// TIA Portal V19 export
DATA_BLOCK "HW_Const_Values"   // DB200
// stored: Access Published, MemoryReserve 100
   VAR
      CU2_PN_IODevice { ExternalAccessible := 'False'; ExternalVisible := 'False'; ExternalWritable := 'False'} : HW_DEVICE := 267;   // "CU2~PN~IODevice"
      CU2_PN { ExternalAccessible := 'False'; ExternalVisible := 'False'; ExternalWritable := 'False'} : HW_INTERFACE := 269;   // "CU2~PN"
      CU2_PN_Port_1 { ExternalAccessible := 'False'; ExternalVisible := 'False'; ExternalWritable := 'False'} : HW_INTERFACE := 270;   // "CU2~PN~Port_1"
      CU2_PN_Port_2 { ExternalAccessible := 'False'; ExternalVisible := 'False'; ExternalWritable := 'False'} : HW_INTERFACE := 271;   // "CU2~PN~Port_2"
      CU2_PN_585A1_ModuleAccessPoint { ExternalAccessible := 'False'; ExternalVisible := 'False'; ExternalWritable := 'False'} : HW_SUBMODULE := 273;   // "CU2~PN~585A1_ModuleAccessPoint"
      CU2_PN_1190A1_ModuleAccessPoint { ExternalAccessible := 'False'; ExternalVisible := 'False'; ExternalWritable := 'False'} : HW_SUBMODULE := 289;   // "CU2~PN~1190A1_ModuleAccessPoint"
      CU2_PN_1300A1_ModuleAccessPoint { ExternalAccessible := 'False'; ExternalVisible := 'False'; ExternalWritable := 'False'} : HW_SUBMODULE := 293;   // "CU2~PN~1300A1_ModuleAccessPoint"
      CU2_PN_830A1_ModuleAccessPoint { ExternalAccessible := 'False'; ExternalVisible := 'False'; ExternalWritable := 'False'} : HW_SUBMODULE := 297;   // "CU2~PN~830A1_ModuleAccessPoint"
      CU2_PN_1 { ExternalAccessible := 'False'; ExternalVisible := 'False'; ExternalWritable := 'False'} : HW_INTERFACE := 269;   // "CU2~PN(1)"
      CU2_PN_Port_1_1 { ExternalAccessible := 'False'; ExternalVisible := 'False'; ExternalWritable := 'False'} : HW_INTERFACE := 270;   // "CU2~PN~Port_1(1)"
      CU2_PN_Port_2_1 { ExternalAccessible := 'False'; ExternalVisible := 'False'; ExternalWritable := 'False'} : HW_INTERFACE := 271;   // "CU2~PN~Port_2(1)"
      CU2_PN_2 { ExternalAccessible := 'False'; ExternalVisible := 'False'; ExternalWritable := 'False'} : HW_INTERFACE := 269;   // "CU2~PN(2)"
      CU2_PN_Port_1_2 { ExternalAccessible := 'False'; ExternalVisible := 'False'; ExternalWritable := 'False'} : HW_INTERFACE := 270;   // "CU2~PN~Port_1(2)"
      CU2_PN_Port_2_2 { ExternalAccessible := 'False'; ExternalVisible := 'False'; ExternalWritable := 'False'} : HW_INTERFACE := 271;   // "CU2~PN~Port_2(2)"
      CU2_PN_3 { ExternalAccessible := 'False'; ExternalVisible := 'False'; ExternalWritable := 'False'} : HW_INTERFACE := 269;   // "CU2~PN(3)"
      CU2_PN_Port_1_3 { ExternalAccessible := 'False'; ExternalVisible := 'False'; ExternalWritable := 'False'} : HW_INTERFACE := 270;   // "CU2~PN~Port_1(3)"
      CU2_PN_Port_2_3 { ExternalAccessible := 'False'; ExternalVisible := 'False'; ExternalWritable := 'False'} : HW_INTERFACE := 271;   // "CU2~PN~Port_2(3)"
      Local_PROFINET_interface_GBIT_3 { ExternalAccessible := 'False'; ExternalVisible := 'False'; ExternalWritable := 'False'} : HW_INTERFACE := 120;   // "Local~PROFINET_interface_GBIT_3"
      Local_PROFINET_interface_GBIT_3_Port_1 { ExternalAccessible := 'False'; ExternalVisible := 'False'; ExternalWritable := 'False'} : HW_INTERFACE := 121;   // "Local~PROFINET_interface_GBIT_3~Port_1"
      Local_412A1 { ExternalAccessible := 'False'; ExternalVisible := 'False'; ExternalWritable := 'False'} : HW_SUBMODULE := 257;   // "Local~412A1"
      Local_413A1 { ExternalAccessible := 'False'; ExternalVisible := 'False'; ExternalWritable := 'False'} : HW_SUBMODULE := 258;   // "Local~413A1"
      Local_413A2 { ExternalAccessible := 'False'; ExternalVisible := 'False'; ExternalWritable := 'False'} : HW_SUBMODULE := 259;   // "Local~413A2"
      Local_414A1 { ExternalAccessible := 'False'; ExternalVisible := 'False'; ExternalWritable := 'False'} : HW_SUBMODULE := 260;   // "Local~414A1"
      Local_415A1 { ExternalAccessible := 'False'; ExternalVisible := 'False'; ExternalWritable := 'False'} : HW_SUBMODULE := 261;   // "Local~415A1"
      Local_415A2 { ExternalAccessible := 'False'; ExternalVisible := 'False'; ExternalWritable := 'False'} : HW_SUBMODULE := 263;   // "Local~415A2"
      HW_460A1_JB001_Proxy { ExternalAccessible := 'False'; ExternalVisible := 'False'; ExternalWritable := 'False'} : HW_SUBMODULE := 302;   // "460A1_JB001~Proxy"
      HW_460A1_JB001_IODevice { ExternalAccessible := 'False'; ExternalVisible := 'False'; ExternalWritable := 'False'} : HW_DEVICE := 300;   // "460A1_JB001~IODevice"
      HW_460A1_JB001_Head { ExternalAccessible := 'False'; ExternalVisible := 'False'; ExternalWritable := 'False'} : HW_SUBMODULE := 303;   // "460A1_JB001~Head"
      HW_460A1_JB001_460A1_X1 { ExternalAccessible := 'False'; ExternalVisible := 'False'; ExternalWritable := 'False'} : HW_INTERFACE := 304;   // "460A1_JB001~460A1_X1"
      HW_460A1_JB001_479A3 { ExternalAccessible := 'False'; ExternalVisible := 'False'; ExternalWritable := 'False'} : HW_SUBMODULE := 355;   // "460A1_JB001~479A3"
      HW_460A1_JB001_479A4 { ExternalAccessible := 'False'; ExternalVisible := 'False'; ExternalWritable := 'False'} : HW_SUBMODULE := 356;   // "460A1_JB001~479A4"
      HW_460A1_JB001_480A1 { ExternalAccessible := 'False'; ExternalVisible := 'False'; ExternalWritable := 'False'} : HW_SUBMODULE := 357;   // "460A1_JB001~480A1"
      HW_460A1_JB001_480A2 { ExternalAccessible := 'False'; ExternalVisible := 'False'; ExternalWritable := 'False'} : HW_SUBMODULE := 358;   // "460A1_JB001~480A2"
      HW_460A1_JB001_482A1 { ExternalAccessible := 'False'; ExternalVisible := 'False'; ExternalWritable := 'False'} : HW_SUBMODULE := 359;   // "460A1_JB001~482A1"
      HW_460A1_JB001_482A2 { ExternalAccessible := 'False'; ExternalVisible := 'False'; ExternalWritable := 'False'} : HW_SUBMODULE := 360;   // "460A1_JB001~482A2"
      HW_460A1_JB001_Server_module_1 { ExternalAccessible := 'False'; ExternalVisible := 'False'; ExternalWritable := 'False'} : HW_SUBMODULE := 456;   // "460A1_JB001~Server_module_1"
      HW_460A1_JB001_464A1 { ExternalAccessible := 'False'; ExternalVisible := 'False'; ExternalWritable := 'False'} : HW_SUBMODULE := 308;   // "460A1_JB001~464A1"
      HW_460A1_JB001_470A2 { ExternalAccessible := 'False'; ExternalVisible := 'False'; ExternalWritable := 'False'} : HW_SUBMODULE := 704;   // "460A1_JB001~470A2"
      HW_460A1_JB001_470A1 { ExternalAccessible := 'False'; ExternalVisible := 'False'; ExternalWritable := 'False'} : HW_SUBMODULE := 703;   // "460A1_JB001~470A1"
      HW_460A1_JB001_463A1 { ExternalAccessible := 'False'; ExternalVisible := 'False'; ExternalWritable := 'False'} : HW_SUBMODULE := 307;   // "460A1_JB001~463A1"
      HW_460A1_JB001_460A1_X1_Port_2 { ExternalAccessible := 'False'; ExternalVisible := 'False'; ExternalWritable := 'False'} : HW_INTERFACE := 306;   // "460A1_JB001~460A1_X1~Port_2"
      HW_460A1_JB001_460A1_X1_Port_1 { ExternalAccessible := 'False'; ExternalVisible := 'False'; ExternalWritable := 'False'} : HW_INTERFACE := 305;   // "460A1_JB001~460A1_X1~Port_1"
      HW_460A1_JB001_465A1 { ExternalAccessible := 'False'; ExternalVisible := 'False'; ExternalWritable := 'False'} : HW_SUBMODULE := 309;   // "460A1_JB001~465A1"
      HW_460A1_JB001_468A1 { ExternalAccessible := 'False'; ExternalVisible := 'False'; ExternalWritable := 'False'} : HW_SUBMODULE := 310;   // "460A1_JB001~468A1"
      HW_460A1_JB001_468A2 { ExternalAccessible := 'False'; ExternalVisible := 'False'; ExternalWritable := 'False'} : HW_SUBMODULE := 311;   // "460A1_JB001~468A2"
      HW_460A1_JB001_468A3 { ExternalAccessible := 'False'; ExternalVisible := 'False'; ExternalWritable := 'False'} : HW_SUBMODULE := 312;   // "460A1_JB001~468A3"
      HW_460A1_JB001_468A4 { ExternalAccessible := 'False'; ExternalVisible := 'False'; ExternalWritable := 'False'} : HW_SUBMODULE := 313;   // "460A1_JB001~468A4"
      HW_460A1_JB001_468A5 { ExternalAccessible := 'False'; ExternalVisible := 'False'; ExternalWritable := 'False'} : HW_SUBMODULE := 314;   // "460A1_JB001~468A5"
      HW_460A1_JB001_468A6 { ExternalAccessible := 'False'; ExternalVisible := 'False'; ExternalWritable := 'False'} : HW_SUBMODULE := 315;   // "460A1_JB001~468A6"
      HW_460A1_JB001_468A7 { ExternalAccessible := 'False'; ExternalVisible := 'False'; ExternalWritable := 'False'} : HW_SUBMODULE := 316;   // "460A1_JB001~468A7"
      HW_460A1_JB001_468A8 { ExternalAccessible := 'False'; ExternalVisible := 'False'; ExternalWritable := 'False'} : HW_SUBMODULE := 317;   // "460A1_JB001~468A8"
      HW_460A1_JB001_471A1 { ExternalAccessible := 'False'; ExternalVisible := 'False'; ExternalWritable := 'False'} : HW_SUBMODULE := 320;   // "460A1_JB001~471A1"
      HW_460A1_JB001_471A2 { ExternalAccessible := 'False'; ExternalVisible := 'False'; ExternalWritable := 'False'} : HW_SUBMODULE := 321;   // "460A1_JB001~471A2"
      HW_460A1_JB001_472A1 { ExternalAccessible := 'False'; ExternalVisible := 'False'; ExternalWritable := 'False'} : HW_SUBMODULE := 322;   // "460A1_JB001~472A1"
      HW_460A1_JB001_474A1 { ExternalAccessible := 'False'; ExternalVisible := 'False'; ExternalWritable := 'False'} : HW_SUBMODULE := 323;   // "460A1_JB001~474A1"
      HW_460A1_JB001_474A2 { ExternalAccessible := 'False'; ExternalVisible := 'False'; ExternalWritable := 'False'} : HW_SUBMODULE := 324;   // "460A1_JB001~474A2"
      HW_460A1_JB001_474A3 { ExternalAccessible := 'False'; ExternalVisible := 'False'; ExternalWritable := 'False'} : HW_SUBMODULE := 325;   // "460A1_JB001~474A3"
      HW_460A1_JB001_474A4 { ExternalAccessible := 'False'; ExternalVisible := 'False'; ExternalWritable := 'False'} : HW_SUBMODULE := 326;   // "460A1_JB001~474A4"
      HW_460A1_JB001_474A5 { ExternalAccessible := 'False'; ExternalVisible := 'False'; ExternalWritable := 'False'} : HW_SUBMODULE := 327;   // "460A1_JB001~474A5"
      HW_460A1_JB001_474A6 { ExternalAccessible := 'False'; ExternalVisible := 'False'; ExternalWritable := 'False'} : HW_SUBMODULE := 328;   // "460A1_JB001~474A6"
      HW_460A1_JB001_474A7 { ExternalAccessible := 'False'; ExternalVisible := 'False'; ExternalWritable := 'False'} : HW_SUBMODULE := 329;   // "460A1_JB001~474A7"
      HW_460A1_JB001_474A8 { ExternalAccessible := 'False'; ExternalVisible := 'False'; ExternalWritable := 'False'} : HW_SUBMODULE := 330;   // "460A1_JB001~474A8"
      HW_460A1_JB001_475A1 { ExternalAccessible := 'False'; ExternalVisible := 'False'; ExternalWritable := 'False'} : HW_SUBMODULE := 331;   // "460A1_JB001~475A1"
      HW_460A1_JB001_475A2 { ExternalAccessible := 'False'; ExternalVisible := 'False'; ExternalWritable := 'False'} : HW_SUBMODULE := 332;   // "460A1_JB001~475A2"
      HW_460A1_JB001_475A3 { ExternalAccessible := 'False'; ExternalVisible := 'False'; ExternalWritable := 'False'} : HW_SUBMODULE := 333;   // "460A1_JB001~475A3"
      HW_460A1_JB001_475A4 { ExternalAccessible := 'False'; ExternalVisible := 'False'; ExternalWritable := 'False'} : HW_SUBMODULE := 334;   // "460A1_JB001~475A4"
      HW_460A1_JB001_475A5 { ExternalAccessible := 'False'; ExternalVisible := 'False'; ExternalWritable := 'False'} : HW_SUBMODULE := 335;   // "460A1_JB001~475A5"
      HW_460A1_JB001_475A6 { ExternalAccessible := 'False'; ExternalVisible := 'False'; ExternalWritable := 'False'} : HW_SUBMODULE := 336;   // "460A1_JB001~475A6"
      HW_460A1_JB001_475A7 { ExternalAccessible := 'False'; ExternalVisible := 'False'; ExternalWritable := 'False'} : HW_SUBMODULE := 337;   // "460A1_JB001~475A7"
      HW_460A1_JB001_475A8 { ExternalAccessible := 'False'; ExternalVisible := 'False'; ExternalWritable := 'False'} : HW_SUBMODULE := 338;   // "460A1_JB001~475A8"
      HW_460A1_JB001_476A1 { ExternalAccessible := 'False'; ExternalVisible := 'False'; ExternalWritable := 'False'} : HW_SUBMODULE := 339;   // "460A1_JB001~476A1"
      HW_460A1_JB001_476A2 { ExternalAccessible := 'False'; ExternalVisible := 'False'; ExternalWritable := 'False'} : HW_SUBMODULE := 340;   // "460A1_JB001~476A2"
      HW_460A1_JB001_476A3 { ExternalAccessible := 'False'; ExternalVisible := 'False'; ExternalWritable := 'False'} : HW_SUBMODULE := 341;   // "460A1_JB001~476A3"
      HW_460A1_JB001_476A4 { ExternalAccessible := 'False'; ExternalVisible := 'False'; ExternalWritable := 'False'} : HW_SUBMODULE := 342;   // "460A1_JB001~476A4"
      HW_460A1_JB001_476A5 { ExternalAccessible := 'False'; ExternalVisible := 'False'; ExternalWritable := 'False'} : HW_SUBMODULE := 343;   // "460A1_JB001~476A5"
      HW_460A1_JB001_476A6 { ExternalAccessible := 'False'; ExternalVisible := 'False'; ExternalWritable := 'False'} : HW_SUBMODULE := 344;   // "460A1_JB001~476A6"
      HW_460A1_JB001_478A1 { ExternalAccessible := 'False'; ExternalVisible := 'False'; ExternalWritable := 'False'} : HW_SUBMODULE := 345;   // "460A1_JB001~478A1"
      HW_460A1_JB001_478A2 { ExternalAccessible := 'False'; ExternalVisible := 'False'; ExternalWritable := 'False'} : HW_SUBMODULE := 346;   // "460A1_JB001~478A2"
      HW_460A1_JB001_478A3 { ExternalAccessible := 'False'; ExternalVisible := 'False'; ExternalWritable := 'False'} : HW_SUBMODULE := 347;   // "460A1_JB001~478A3"
      HW_460A1_JB001_478A4 { ExternalAccessible := 'False'; ExternalVisible := 'False'; ExternalWritable := 'False'} : HW_SUBMODULE := 348;   // "460A1_JB001~478A4"
      HW_460A1_JB001_478A5 { ExternalAccessible := 'False'; ExternalVisible := 'False'; ExternalWritable := 'False'} : HW_SUBMODULE := 349;   // "460A1_JB001~478A5"
      HW_460A1_JB001_478A6 { ExternalAccessible := 'False'; ExternalVisible := 'False'; ExternalWritable := 'False'} : HW_SUBMODULE := 350;   // "460A1_JB001~478A6"
      HW_460A1_JB001_478A7 { ExternalAccessible := 'False'; ExternalVisible := 'False'; ExternalWritable := 'False'} : HW_SUBMODULE := 351;   // "460A1_JB001~478A7"
      HW_460A1_JB001_478A8 { ExternalAccessible := 'False'; ExternalVisible := 'False'; ExternalWritable := 'False'} : HW_SUBMODULE := 352;   // "460A1_JB001~478A8"
      HW_460A1_JB001_479A1 { ExternalAccessible := 'False'; ExternalVisible := 'False'; ExternalWritable := 'False'} : HW_SUBMODULE := 353;   // "460A1_JB001~479A1"
      HW_460A1_JB001_479A2 { ExternalAccessible := 'False'; ExternalVisible := 'False'; ExternalWritable := 'False'} : HW_SUBMODULE := 354;   // "460A1_JB001~479A2"
      HW_490A1_JB301_Proxy { ExternalAccessible := 'False'; ExternalVisible := 'False'; ExternalWritable := 'False'} : HW_SUBMODULE := 363;   // "490A1_JB301~Proxy"
      HW_490A1_JB301_IODevice { ExternalAccessible := 'False'; ExternalVisible := 'False'; ExternalWritable := 'False'} : HW_DEVICE := 361;   // "490A1_JB301~IODevice"
      HW_490A1_JB301_Head { ExternalAccessible := 'False'; ExternalVisible := 'False'; ExternalWritable := 'False'} : HW_SUBMODULE := 364;   // "490A1_JB301~Head"
      HW_490A1_JB301_PROFINET_interface { ExternalAccessible := 'False'; ExternalVisible := 'False'; ExternalWritable := 'False'} : HW_INTERFACE := 365;   // "490A1_JB301~PROFINET_interface"
      HW_490A1_JB301_495A2 { ExternalAccessible := 'False'; ExternalVisible := 'False'; ExternalWritable := 'False'} : HW_SUBMODULE := 369;   // "490A1_JB301~495A2"
      HW_490A1_JB301_495A1 { ExternalAccessible := 'False'; ExternalVisible := 'False'; ExternalWritable := 'False'} : HW_SUBMODULE := 368;   // "490A1_JB301~495A1"
      HW_490A1_JB301_PROFINET_interface_Port_2 { ExternalAccessible := 'False'; ExternalVisible := 'False'; ExternalWritable := 'False'} : HW_INTERFACE := 367;   // "490A1_JB301~PROFINET_interface~Port_2"
      HW_490A1_JB301_PROFINET_interface_Port_1 { ExternalAccessible := 'False'; ExternalVisible := 'False'; ExternalWritable := 'False'} : HW_INTERFACE := 366;   // "490A1_JB301~PROFINET_interface~Port_1"
      HW_510A1_JB302_Proxy { ExternalAccessible := 'False'; ExternalVisible := 'False'; ExternalWritable := 'False'} : HW_SUBMODULE := 378;   // "510A1_JB302~Proxy"
      HW_510A1_JB302_IODevice { ExternalAccessible := 'False'; ExternalVisible := 'False'; ExternalWritable := 'False'} : HW_DEVICE := 376;   // "510A1_JB302~IODevice"
      HW_510A1_JB302_Head { ExternalAccessible := 'False'; ExternalVisible := 'False'; ExternalWritable := 'False'} : HW_SUBMODULE := 379;   // "510A1_JB302~Head"
      HW_510A1_JB302_PROFINET_interface { ExternalAccessible := 'False'; ExternalVisible := 'False'; ExternalWritable := 'False'} : HW_INTERFACE := 380;   // "510A1_JB302~PROFINET_interface"
      HW_510A1_JB302_515A2 { ExternalAccessible := 'False'; ExternalVisible := 'False'; ExternalWritable := 'False'} : HW_SUBMODULE := 386;   // "510A1_JB302~515A2"
      HW_510A1_JB302_515A1 { ExternalAccessible := 'False'; ExternalVisible := 'False'; ExternalWritable := 'False'} : HW_SUBMODULE := 385;   // "510A1_JB302~515A1"
      HW_510A1_JB302_513A1 { ExternalAccessible := 'False'; ExternalVisible := 'False'; ExternalWritable := 'False'} : HW_SUBMODULE := 384;   // "510A1_JB302~513A1"
      HW_510A1_JB302_512A1 { ExternalAccessible := 'False'; ExternalVisible := 'False'; ExternalWritable := 'False'} : HW_SUBMODULE := 383;   // "510A1_JB302~512A1"
      HW_510A1_JB302_PROFINET_interface_Port_2 { ExternalAccessible := 'False'; ExternalVisible := 'False'; ExternalWritable := 'False'} : HW_INTERFACE := 382;   // "510A1_JB302~PROFINET_interface~Port_2"
      HW_510A1_JB302_PROFINET_interface_Port_1 { ExternalAccessible := 'False'; ExternalVisible := 'False'; ExternalWritable := 'False'} : HW_INTERFACE := 381;   // "510A1_JB302~PROFINET_interface~Port_1"
      HW_530A1_JB305_Proxy { ExternalAccessible := 'False'; ExternalVisible := 'False'; ExternalWritable := 'False'} : HW_SUBMODULE := 413;   // "530A1_JB305~Proxy"
      HW_530A1_JB305_IODevice { ExternalAccessible := 'False'; ExternalVisible := 'False'; ExternalWritable := 'False'} : HW_DEVICE := 411;   // "530A1_JB305~IODevice"
      HW_530A1_JB305_Head { ExternalAccessible := 'False'; ExternalVisible := 'False'; ExternalWritable := 'False'} : HW_SUBMODULE := 414;   // "530A1_JB305~Head"
      HW_530A1_JB305_PROFINET_interface { ExternalAccessible := 'False'; ExternalVisible := 'False'; ExternalWritable := 'False'} : HW_INTERFACE := 415;   // "530A1_JB305~PROFINET_interface"
      HW_530A1_JB305_542A3 { ExternalAccessible := 'False'; ExternalVisible := 'False'; ExternalWritable := 'False'} : HW_SUBMODULE := 434;   // "530A1_JB305~542A3"
      HW_530A1_JB305_542A2 { ExternalAccessible := 'False'; ExternalVisible := 'False'; ExternalWritable := 'False'} : HW_SUBMODULE := 433;   // "530A1_JB305~542A2"
      HW_530A1_JB305_542A1 { ExternalAccessible := 'False'; ExternalVisible := 'False'; ExternalWritable := 'False'} : HW_SUBMODULE := 432;   // "530A1_JB305~542A1"
      HW_530A1_JB305_540A2 { ExternalAccessible := 'False'; ExternalVisible := 'False'; ExternalWritable := 'False'} : HW_SUBMODULE := 431;   // "530A1_JB305~540A2"
      HW_530A1_JB305_540A1 { ExternalAccessible := 'False'; ExternalVisible := 'False'; ExternalWritable := 'False'} : HW_SUBMODULE := 430;   // "530A1_JB305~540A1"
      HW_530A1_JB305_538A6 { ExternalAccessible := 'False'; ExternalVisible := 'False'; ExternalWritable := 'False'} : HW_SUBMODULE := 429;   // "530A1_JB305~538A6"
      HW_530A1_JB305_538A5 { ExternalAccessible := 'False'; ExternalVisible := 'False'; ExternalWritable := 'False'} : HW_SUBMODULE := 428;   // "530A1_JB305~538A5"
      HW_530A1_JB305_538A4 { ExternalAccessible := 'False'; ExternalVisible := 'False'; ExternalWritable := 'False'} : HW_SUBMODULE := 427;   // "530A1_JB305~538A4"
      HW_530A1_JB305_538A3 { ExternalAccessible := 'False'; ExternalVisible := 'False'; ExternalWritable := 'False'} : HW_SUBMODULE := 426;   // "530A1_JB305~538A3"
      HW_530A1_JB305_538A2 { ExternalAccessible := 'False'; ExternalVisible := 'False'; ExternalWritable := 'False'} : HW_SUBMODULE := 425;   // "530A1_JB305~538A2"
      HW_530A1_JB305_538A1 { ExternalAccessible := 'False'; ExternalVisible := 'False'; ExternalWritable := 'False'} : HW_SUBMODULE := 424;   // "530A1_JB305~538A1"
      HW_530A1_JB305_537A1 { ExternalAccessible := 'False'; ExternalVisible := 'False'; ExternalWritable := 'False'} : HW_SUBMODULE := 423;   // "530A1_JB305~537A1"
      HW_530A1_JB305_536A1 { ExternalAccessible := 'False'; ExternalVisible := 'False'; ExternalWritable := 'False'} : HW_SUBMODULE := 422;   // "530A1_JB305~536A1"
      HW_530A1_JB305_535A2 { ExternalAccessible := 'False'; ExternalVisible := 'False'; ExternalWritable := 'False'} : HW_SUBMODULE := 421;   // "530A1_JB305~535A2"
      HW_530A1_JB305_535A1 { ExternalAccessible := 'False'; ExternalVisible := 'False'; ExternalWritable := 'False'} : HW_SUBMODULE := 420;   // "530A1_JB305~535A1"
      HW_530A1_JB305_533A1 { ExternalAccessible := 'False'; ExternalVisible := 'False'; ExternalWritable := 'False'} : HW_SUBMODULE := 419;   // "530A1_JB305~533A1"
      HW_530A1_JB305_PROFINET_interface_Port_2 { ExternalAccessible := 'False'; ExternalVisible := 'False'; ExternalWritable := 'False'} : HW_INTERFACE := 417;   // "530A1_JB305~PROFINET_interface~Port_2"
      HW_530A1_JB305_PROFINET_interface_Port_1 { ExternalAccessible := 'False'; ExternalVisible := 'False'; ExternalWritable := 'False'} : HW_INTERFACE := 416;   // "530A1_JB305~PROFINET_interface~Port_1"
      HW_550A1_JB306_Proxy { ExternalAccessible := 'False'; ExternalVisible := 'False'; ExternalWritable := 'False'} : HW_SUBMODULE := 437;   // "550A1_JB306~Proxy"
      HW_550A1_JB306_IODevice { ExternalAccessible := 'False'; ExternalVisible := 'False'; ExternalWritable := 'False'} : HW_DEVICE := 435;   // "550A1_JB306~IODevice"
      HW_550A1_JB306_Head { ExternalAccessible := 'False'; ExternalVisible := 'False'; ExternalWritable := 'False'} : HW_SUBMODULE := 438;   // "550A1_JB306~Head"
      HW_550A1_JB306_PROFINET_interface { ExternalAccessible := 'False'; ExternalVisible := 'False'; ExternalWritable := 'False'} : HW_INTERFACE := 439;   // "550A1_JB306~PROFINET_interface"
      HW_550A1_JB306_562A3 { ExternalAccessible := 'False'; ExternalVisible := 'False'; ExternalWritable := 'False'} : HW_SUBMODULE := 455;   // "550A1_JB306~562A3"
      HW_550A1_JB306_562A2 { ExternalAccessible := 'False'; ExternalVisible := 'False'; ExternalWritable := 'False'} : HW_SUBMODULE := 454;   // "550A1_JB306~562A2"
      HW_550A1_JB306_562A1 { ExternalAccessible := 'False'; ExternalVisible := 'False'; ExternalWritable := 'False'} : HW_SUBMODULE := 453;   // "550A1_JB306~562A1"
      HW_550A1_JB306_560A2 { ExternalAccessible := 'False'; ExternalVisible := 'False'; ExternalWritable := 'False'} : HW_SUBMODULE := 452;   // "550A1_JB306~560A2"
      HW_550A1_JB306_560A1 { ExternalAccessible := 'False'; ExternalVisible := 'False'; ExternalWritable := 'False'} : HW_SUBMODULE := 451;   // "550A1_JB306~560A1"
      HW_550A1_JB306_558A6 { ExternalAccessible := 'False'; ExternalVisible := 'False'; ExternalWritable := 'False'} : HW_SUBMODULE := 450;   // "550A1_JB306~558A6"
      HW_550A1_JB306_558A5 { ExternalAccessible := 'False'; ExternalVisible := 'False'; ExternalWritable := 'False'} : HW_SUBMODULE := 449;   // "550A1_JB306~558A5"
      HW_550A1_JB306_558A4 { ExternalAccessible := 'False'; ExternalVisible := 'False'; ExternalWritable := 'False'} : HW_SUBMODULE := 448;   // "550A1_JB306~558A4"
      HW_550A1_JB306_558A3 { ExternalAccessible := 'False'; ExternalVisible := 'False'; ExternalWritable := 'False'} : HW_SUBMODULE := 447;   // "550A1_JB306~558A3"
      HW_550A1_JB306_558A2 { ExternalAccessible := 'False'; ExternalVisible := 'False'; ExternalWritable := 'False'} : HW_SUBMODULE := 446;   // "550A1_JB306~558A2"
      HW_550A1_JB306_558A1 { ExternalAccessible := 'False'; ExternalVisible := 'False'; ExternalWritable := 'False'} : HW_SUBMODULE := 445;   // "550A1_JB306~558A1"
      HW_550A1_JB306_556A1 { ExternalAccessible := 'False'; ExternalVisible := 'False'; ExternalWritable := 'False'} : HW_SUBMODULE := 444;   // "550A1_JB306~556A1"
      HW_550A1_JB306_555A1 { ExternalAccessible := 'False'; ExternalVisible := 'False'; ExternalWritable := 'False'} : HW_SUBMODULE := 443;   // "550A1_JB306~555A1"
      HW_550A1_JB306_552A1 { ExternalAccessible := 'False'; ExternalVisible := 'False'; ExternalWritable := 'False'} : HW_SUBMODULE := 442;   // "550A1_JB306~552A1"
      HW_550A1_JB306_PROFINET_interface_Port_2 { ExternalAccessible := 'False'; ExternalVisible := 'False'; ExternalWritable := 'False'} : HW_INTERFACE := 441;   // "550A1_JB306~PROFINET_interface~Port_2"
      HW_550A1_JB306_PROFINET_interface_Port_1 { ExternalAccessible := 'False'; ExternalVisible := 'False'; ExternalWritable := 'False'} : HW_INTERFACE := 440;   // "550A1_JB306~PROFINET_interface~Port_1"
      CU1_PN_IODevice { ExternalAccessible := 'False'; ExternalVisible := 'False'; ExternalWritable := 'False'} : HW_DEVICE := 275;   // "CU1~PN~IODevice"
      CU1_PN { ExternalAccessible := 'False'; ExternalVisible := 'False'; ExternalWritable := 'False'} : HW_INTERFACE := 277;   // "CU1~PN"
      CU1_PN_Port_1 { ExternalAccessible := 'False'; ExternalVisible := 'False'; ExternalWritable := 'False'} : HW_INTERFACE := 278;   // "CU1~PN~Port_1"
      CU1_PN_Port_2 { ExternalAccessible := 'False'; ExternalVisible := 'False'; ExternalWritable := 'False'} : HW_INTERFACE := 279;   // "CU1~PN~Port_2"
      CU1_PN_580A1_ModuleAccessPoint { ExternalAccessible := 'False'; ExternalVisible := 'False'; ExternalWritable := 'False'} : HW_SUBMODULE := 281;   // "CU1~PN~580A1_ModuleAccessPoint"
      CU1_PN_740A1_1_ModuleAccessPoint { ExternalAccessible := 'False'; ExternalVisible := 'False'; ExternalWritable := 'False'} : HW_SUBMODULE := 284;   // "CU1~PN~740A1_1_ModuleAccessPoint"
      CU1_PN_740A1_2_ModuleAccessPoint { ExternalAccessible := 'False'; ExternalVisible := 'False'; ExternalWritable := 'False'} : HW_SUBMODULE := 318;   // "CU1~PN~740A1_2_ModuleAccessPoint"
      CU1_PN_690A1_1_ModuleAccessPoint { ExternalAccessible := 'False'; ExternalVisible := 'False'; ExternalWritable := 'False'} : HW_SUBMODULE := 459;   // "CU1~PN~690A1_1_ModuleAccessPoint"
      CU1_PN_690A1_2_ModuleAccessPoint { ExternalAccessible := 'False'; ExternalVisible := 'False'; ExternalWritable := 'False'} : HW_SUBMODULE := 463;   // "CU1~PN~690A1_2_ModuleAccessPoint"
      CU1_PN_890A1_1_ModuleAccessPoint { ExternalAccessible := 'False'; ExternalVisible := 'False'; ExternalWritable := 'False'} : HW_SUBMODULE := 467;   // "CU1~PN~890A1_1_ModuleAccessPoint"
      CU1_PN_890A1_2_ModuleAccessPoint { ExternalAccessible := 'False'; ExternalVisible := 'False'; ExternalWritable := 'False'} : HW_SUBMODULE := 471;   // "CU1~PN~890A1_2_ModuleAccessPoint"
      CU1_PN_1 { ExternalAccessible := 'False'; ExternalVisible := 'False'; ExternalWritable := 'False'} : HW_INTERFACE := 277;   // "CU1~PN(1)"
      CU1_PN_Port_1_1 { ExternalAccessible := 'False'; ExternalVisible := 'False'; ExternalWritable := 'False'} : HW_INTERFACE := 278;   // "CU1~PN~Port_1(1)"
      CU1_PN_Port_2_1 { ExternalAccessible := 'False'; ExternalVisible := 'False'; ExternalWritable := 'False'} : HW_INTERFACE := 279;   // "CU1~PN~Port_2(1)"
      CU1_PN_2 { ExternalAccessible := 'False'; ExternalVisible := 'False'; ExternalWritable := 'False'} : HW_INTERFACE := 277;   // "CU1~PN(2)"
      CU1_PN_Port_1_2 { ExternalAccessible := 'False'; ExternalVisible := 'False'; ExternalWritable := 'False'} : HW_INTERFACE := 278;   // "CU1~PN~Port_1(2)"
      CU1_PN_Port_2_2 { ExternalAccessible := 'False'; ExternalVisible := 'False'; ExternalWritable := 'False'} : HW_INTERFACE := 279;   // "CU1~PN~Port_2(2)"
      CU1_PN_3 { ExternalAccessible := 'False'; ExternalVisible := 'False'; ExternalWritable := 'False'} : HW_INTERFACE := 277;   // "CU1~PN(3)"
      CU1_PN_Port_1_3 { ExternalAccessible := 'False'; ExternalVisible := 'False'; ExternalWritable := 'False'} : HW_INTERFACE := 278;   // "CU1~PN~Port_1(3)"
      CU1_PN_Port_2_3 { ExternalAccessible := 'False'; ExternalVisible := 'False'; ExternalWritable := 'False'} : HW_INTERFACE := 279;   // "CU1~PN~Port_2(3)"
      CU3_PROFINET_interface_IODevice { ExternalAccessible := 'False'; ExternalVisible := 'False'; ExternalWritable := 'False'} : HW_DEVICE := 475;   // "CU3~PROFINET_interface~IODevice"
      CU3_PROFINET_interface { ExternalAccessible := 'False'; ExternalVisible := 'False'; ExternalWritable := 'False'} : HW_INTERFACE := 477;   // "CU3~PROFINET_interface"
      CU3_PROFINET_interface_Port_1 { ExternalAccessible := 'False'; ExternalVisible := 'False'; ExternalWritable := 'False'} : HW_INTERFACE := 478;   // "CU3~PROFINET_interface~Port_1"
      CU3_PROFINET_interface_Port_2 { ExternalAccessible := 'False'; ExternalVisible := 'False'; ExternalWritable := 'False'} : HW_INTERFACE := 479;   // "CU3~PROFINET_interface~Port_2"
      CU3_PROFINET_interface_590A1_ModuleAccessPoint { ExternalAccessible := 'False'; ExternalVisible := 'False'; ExternalWritable := 'False'} : HW_SUBMODULE := 481;   // "CU3~PROFINET_interface~590A1_ModuleAccessPoint"
      CU3_PROFINET_interface_590A1_SIEMENS_telegram_393 { ExternalAccessible := 'False'; ExternalVisible := 'False'; ExternalWritable := 'False'} : HW_SUBMODULE := 482;   // "CU3~PROFINET_interface~590A1_SIEMENS_telegram_393"
      CU3_PROFINET_interface_1410A1_1_ModuleAccessPoint { ExternalAccessible := 'False'; ExternalVisible := 'False'; ExternalWritable := 'False'} : HW_SUBMODULE := 484;   // "CU3~PROFINET_interface~1410A1_1_ModuleAccessPoint"
      CU3_PROFINET_interface_1410A1_1_PROFIsafe_telegram_30 { ExternalAccessible := 'False'; ExternalVisible := 'False'; ExternalWritable := 'False'} : HW_SUBMODULE := 486;   // "CU3~PROFINET_interface~1410A1_1_PROFIsafe_telegram_30"
      CU3_PROFINET_interface_1410A1_2_ModuleAccessPoint { ExternalAccessible := 'False'; ExternalVisible := 'False'; ExternalWritable := 'False'} : HW_SUBMODULE := 488;   // "CU3~PROFINET_interface~1410A1_2_ModuleAccessPoint"
      CU3_PROFINET_interface_1410A1_2_PROFIsafe_telegram_30 { ExternalAccessible := 'False'; ExternalVisible := 'False'; ExternalWritable := 'False'} : HW_SUBMODULE := 490;   // "CU3~PROFINET_interface~1410A1_2_PROFIsafe_telegram_30"
      CU3_PROFINET_interface_1430A1_1_ModuleAccessPoint { ExternalAccessible := 'False'; ExternalVisible := 'False'; ExternalWritable := 'False'} : HW_SUBMODULE := 492;   // "CU3~PROFINET_interface~1430A1_1_ModuleAccessPoint"
      CU3_PROFINET_interface_1430A1_1_PROFIsafe_telegram_30 { ExternalAccessible := 'False'; ExternalVisible := 'False'; ExternalWritable := 'False'} : HW_SUBMODULE := 494;   // "CU3~PROFINET_interface~1430A1_1_PROFIsafe_telegram_30"
      CU3_PROFINET_interface_1430A1_2_ModuleAccessPoint { ExternalAccessible := 'False'; ExternalVisible := 'False'; ExternalWritable := 'False'} : HW_SUBMODULE := 496;   // "CU3~PROFINET_interface~1430A1_2_ModuleAccessPoint"
      CU3_PROFINET_interface_1430A1_2_PROFIsafe_telegram_30 { ExternalAccessible := 'False'; ExternalVisible := 'False'; ExternalWritable := 'False'} : HW_SUBMODULE := 498;   // "CU3~PROFINET_interface~1430A1_2_PROFIsafe_telegram_30"
      CU3_PROFINET_interface_1260A1_1_ModuleAccessPoint { ExternalAccessible := 'False'; ExternalVisible := 'False'; ExternalWritable := 'False'} : HW_SUBMODULE := 500;   // "CU3~PROFINET_interface~1260A1_1_ModuleAccessPoint"
      CU3_PROFINET_interface_1260A1_1_PROFIsafe_telegram_30 { ExternalAccessible := 'False'; ExternalVisible := 'False'; ExternalWritable := 'False'} : HW_SUBMODULE := 502;   // "CU3~PROFINET_interface~1260A1_1_PROFIsafe_telegram_30"
      CU3_PROFINET_interface_1260A1_2_ModuleAccessPoint { ExternalAccessible := 'False'; ExternalVisible := 'False'; ExternalWritable := 'False'} : HW_SUBMODULE := 504;   // "CU3~PROFINET_interface~1260A1_2_ModuleAccessPoint"
      CU3_PROFINET_interface_1260A1_2_PROFIsafe_telegram_30 { ExternalAccessible := 'False'; ExternalVisible := 'False'; ExternalWritable := 'False'} : HW_SUBMODULE := 506;   // "CU3~PROFINET_interface~1260A1_2_PROFIsafe_telegram_30"
      CU3_PROFINET_interface_1 { ExternalAccessible := 'False'; ExternalVisible := 'False'; ExternalWritable := 'False'} : HW_INTERFACE := 477;   // "CU3~PROFINET_interface(1)"
      CU3_PROFINET_interface_Port_1_1 { ExternalAccessible := 'False'; ExternalVisible := 'False'; ExternalWritable := 'False'} : HW_INTERFACE := 478;   // "CU3~PROFINET_interface~Port_1(1)"
      CU3_PROFINET_interface_Port_2_1 { ExternalAccessible := 'False'; ExternalVisible := 'False'; ExternalWritable := 'False'} : HW_INTERFACE := 479;   // "CU3~PROFINET_interface~Port_2(1)"
      CU3_PROFINET_interface_2 { ExternalAccessible := 'False'; ExternalVisible := 'False'; ExternalWritable := 'False'} : HW_INTERFACE := 477;   // "CU3~PROFINET_interface(2)"
      CU3_PROFINET_interface_Port_1_2 { ExternalAccessible := 'False'; ExternalVisible := 'False'; ExternalWritable := 'False'} : HW_INTERFACE := 478;   // "CU3~PROFINET_interface~Port_1(2)"
      CU3_PROFINET_interface_Port_2_2 { ExternalAccessible := 'False'; ExternalVisible := 'False'; ExternalWritable := 'False'} : HW_INTERFACE := 479;   // "CU3~PROFINET_interface~Port_2(2)"
      CU3_PROFINET_interface_3 { ExternalAccessible := 'False'; ExternalVisible := 'False'; ExternalWritable := 'False'} : HW_INTERFACE := 477;   // "CU3~PROFINET_interface(3)"
      CU3_PROFINET_interface_Port_1_3 { ExternalAccessible := 'False'; ExternalVisible := 'False'; ExternalWritable := 'False'} : HW_INTERFACE := 478;   // "CU3~PROFINET_interface~Port_1(3)"
      CU3_PROFINET_interface_Port_2_3 { ExternalAccessible := 'False'; ExternalVisible := 'False'; ExternalWritable := 'False'} : HW_INTERFACE := 479;   // "CU3~PROFINET_interface~Port_2(3)"
      CU4_PN_IODevice { ExternalAccessible := 'False'; ExternalVisible := 'False'; ExternalWritable := 'False'} : HW_DEVICE := 508;   // "CU4~PN~IODevice"
      CU4_PN { ExternalAccessible := 'False'; ExternalVisible := 'False'; ExternalWritable := 'False'} : HW_INTERFACE := 510;   // "CU4~PN"
      CU4_PN_Port_1 { ExternalAccessible := 'False'; ExternalVisible := 'False'; ExternalWritable := 'False'} : HW_INTERFACE := 511;   // "CU4~PN~Port_1"
      CU4_PN_Port_2 { ExternalAccessible := 'False'; ExternalVisible := 'False'; ExternalWritable := 'False'} : HW_INTERFACE := 512;   // "CU4~PN~Port_2"
      CU4_PN_595A1_ModuleAccessPoint { ExternalAccessible := 'False'; ExternalVisible := 'False'; ExternalWritable := 'False'} : HW_SUBMODULE := 514;   // "CU4~PN~595A1_ModuleAccessPoint"
      CU4_PN_595A1_SIEMENS_telegram_393 { ExternalAccessible := 'False'; ExternalVisible := 'False'; ExternalWritable := 'False'} : HW_SUBMODULE := 515;   // "CU4~PN~595A1_SIEMENS_telegram_393"
      CU4_PN_980A1_1_ModuleAccessPoint { ExternalAccessible := 'False'; ExternalVisible := 'False'; ExternalWritable := 'False'} : HW_SUBMODULE := 517;   // "CU4~PN~980A1_1_ModuleAccessPoint"
      CU4_PN_980A1_1_PROFIsafe_telegram_30 { ExternalAccessible := 'False'; ExternalVisible := 'False'; ExternalWritable := 'False'} : HW_SUBMODULE := 519;   // "CU4~PN~980A1_1_PROFIsafe_telegram_30"
      CU4_PN_980A1_2_ModuleAccessPoint { ExternalAccessible := 'False'; ExternalVisible := 'False'; ExternalWritable := 'False'} : HW_SUBMODULE := 521;   // "CU4~PN~980A1_2_ModuleAccessPoint"
      CU4_PN_980A1_2_PROFIsafe_telegram_30 { ExternalAccessible := 'False'; ExternalVisible := 'False'; ExternalWritable := 'False'} : HW_SUBMODULE := 523;   // "CU4~PN~980A1_2_PROFIsafe_telegram_30"
      CU4_PN_1030A1_1_ModuleAccessPoint { ExternalAccessible := 'False'; ExternalVisible := 'False'; ExternalWritable := 'False'} : HW_SUBMODULE := 525;   // "CU4~PN~1030A1_1_ModuleAccessPoint"
      CU4_PN_1030A1_1_PROFIsafe_telegram_30 { ExternalAccessible := 'False'; ExternalVisible := 'False'; ExternalWritable := 'False'} : HW_SUBMODULE := 527;   // "CU4~PN~1030A1_1_PROFIsafe_telegram_30"
      CU4_PN_1030A1_2_ModuleAccessPoint { ExternalAccessible := 'False'; ExternalVisible := 'False'; ExternalWritable := 'False'} : HW_SUBMODULE := 529;   // "CU4~PN~1030A1_2_ModuleAccessPoint"
      CU4_PN_1030A1_2_PROFIsafe_telegram_30 { ExternalAccessible := 'False'; ExternalVisible := 'False'; ExternalWritable := 'False'} : HW_SUBMODULE := 531;   // "CU4~PN~1030A1_2_PROFIsafe_telegram_30"
      CU4_PN_1070A1_1_ModuleAccessPoint { ExternalAccessible := 'False'; ExternalVisible := 'False'; ExternalWritable := 'False'} : HW_SUBMODULE := 533;   // "CU4~PN~1070A1_1_ModuleAccessPoint"
      CU4_PN_1070A1_1_PROFIsafe_telegram_30 { ExternalAccessible := 'False'; ExternalVisible := 'False'; ExternalWritable := 'False'} : HW_SUBMODULE := 535;   // "CU4~PN~1070A1_1_PROFIsafe_telegram_30"
      CU4_PN_1070A1_2_ModuleAccessPoint { ExternalAccessible := 'False'; ExternalVisible := 'False'; ExternalWritable := 'False'} : HW_SUBMODULE := 537;   // "CU4~PN~1070A1_2_ModuleAccessPoint"
      CU4_PN_1070A1_2_PROFIsafe_telegram_30 { ExternalAccessible := 'False'; ExternalVisible := 'False'; ExternalWritable := 'False'} : HW_SUBMODULE := 539;   // "CU4~PN~1070A1_2_PROFIsafe_telegram_30"
      CU4_PN_1 { ExternalAccessible := 'False'; ExternalVisible := 'False'; ExternalWritable := 'False'} : HW_INTERFACE := 510;   // "CU4~PN(1)"
      CU4_PN_Port_1_1 { ExternalAccessible := 'False'; ExternalVisible := 'False'; ExternalWritable := 'False'} : HW_INTERFACE := 511;   // "CU4~PN~Port_1(1)"
      CU4_PN_Port_2_1 { ExternalAccessible := 'False'; ExternalVisible := 'False'; ExternalWritable := 'False'} : HW_INTERFACE := 512;   // "CU4~PN~Port_2(1)"
      CU4_PN_2 { ExternalAccessible := 'False'; ExternalVisible := 'False'; ExternalWritable := 'False'} : HW_INTERFACE := 510;   // "CU4~PN(2)"
      CU4_PN_Port_1_2 { ExternalAccessible := 'False'; ExternalVisible := 'False'; ExternalWritable := 'False'} : HW_INTERFACE := 511;   // "CU4~PN~Port_1(2)"
      CU4_PN_Port_2_2 { ExternalAccessible := 'False'; ExternalVisible := 'False'; ExternalWritable := 'False'} : HW_INTERFACE := 512;   // "CU4~PN~Port_2(2)"
      CU4_PN_3 { ExternalAccessible := 'False'; ExternalVisible := 'False'; ExternalWritable := 'False'} : HW_INTERFACE := 510;   // "CU4~PN(3)"
      CU4_PN_Port_1_3 { ExternalAccessible := 'False'; ExternalVisible := 'False'; ExternalWritable := 'False'} : HW_INTERFACE := 511;   // "CU4~PN~Port_1(3)"
      CU4_PN_Port_2_3 { ExternalAccessible := 'False'; ExternalVisible := 'False'; ExternalWritable := 'False'} : HW_INTERFACE := 512;   // "CU4~PN~Port_2(3)"
      CU5_PN_IODevice { ExternalAccessible := 'False'; ExternalVisible := 'False'; ExternalWritable := 'False'} : HW_DEVICE := 541;   // "CU5~PN~IODevice"
      CU5_PN { ExternalAccessible := 'False'; ExternalVisible := 'False'; ExternalWritable := 'False'} : HW_INTERFACE := 543;   // "CU5~PN"
      CU5_PN_Port_1 { ExternalAccessible := 'False'; ExternalVisible := 'False'; ExternalWritable := 'False'} : HW_INTERFACE := 544;   // "CU5~PN~Port_1"
      CU5_PN_Port_2 { ExternalAccessible := 'False'; ExternalVisible := 'False'; ExternalWritable := 'False'} : HW_INTERFACE := 545;   // "CU5~PN~Port_2"
      CU5_PN_600A1_ModuleAccessPoint { ExternalAccessible := 'False'; ExternalVisible := 'False'; ExternalWritable := 'False'} : HW_SUBMODULE := 547;   // "CU5~PN~600A1_ModuleAccessPoint"
      CU5_PN_600A1_SIEMENS_telegram_393 { ExternalAccessible := 'False'; ExternalVisible := 'False'; ExternalWritable := 'False'} : HW_SUBMODULE := 548;   // "CU5~PN~600A1_SIEMENS_telegram_393"
      CU5_PN_1950A1_ModuleAccessPoint { ExternalAccessible := 'False'; ExternalVisible := 'False'; ExternalWritable := 'False'} : HW_SUBMODULE := 550;   // "CU5~PN~1950A1_ModuleAccessPoint"
      CU5_PN_1950A1_SIEMENS_telegram_111 { ExternalAccessible := 'False'; ExternalVisible := 'False'; ExternalWritable := 'False'} : HW_SUBMODULE := 551;   // "CU5~PN~1950A1_SIEMENS_telegram_111"
      CU5_PN_1950A1_PROFIsafe_telegram_30 { ExternalAccessible := 'False'; ExternalVisible := 'False'; ExternalWritable := 'False'} : HW_SUBMODULE := 552;   // "CU5~PN~1950A1_PROFIsafe_telegram_30"
      CU5_PN_1480A1_1_ModuleAccessPoint { ExternalAccessible := 'False'; ExternalVisible := 'False'; ExternalWritable := 'False'} : HW_SUBMODULE := 554;   // "CU5~PN~1480A1_1_ModuleAccessPoint"
      CU5_PN_1480A1_1_PROFIsafe_telegram_30 { ExternalAccessible := 'False'; ExternalVisible := 'False'; ExternalWritable := 'False'} : HW_SUBMODULE := 556;   // "CU5~PN~1480A1_1_PROFIsafe_telegram_30"
      CU5_PN_1480A1_2_ModuleAccessPoint { ExternalAccessible := 'False'; ExternalVisible := 'False'; ExternalWritable := 'False'} : HW_SUBMODULE := 558;   // "CU5~PN~1480A1_2_ModuleAccessPoint"
      CU5_PN_1480A1_2_PROFIsafe_telegram_30 { ExternalAccessible := 'False'; ExternalVisible := 'False'; ExternalWritable := 'False'} : HW_SUBMODULE := 560;   // "CU5~PN~1480A1_2_PROFIsafe_telegram_30"
      CU5_PN_1560A1_1_ModuleAccessPoint { ExternalAccessible := 'False'; ExternalVisible := 'False'; ExternalWritable := 'False'} : HW_SUBMODULE := 562;   // "CU5~PN~1560A1_1_ModuleAccessPoint"
      CU5_PN_1560A1_1_SIEMENS_telegram_111 { ExternalAccessible := 'False'; ExternalVisible := 'False'; ExternalWritable := 'False'} : HW_SUBMODULE := 563;   // "CU5~PN~1560A1_1_SIEMENS_telegram_111"
      CU5_PN_1560A1_1_PROFIsafe_telegram_30 { ExternalAccessible := 'False'; ExternalVisible := 'False'; ExternalWritable := 'False'} : HW_SUBMODULE := 564;   // "CU5~PN~1560A1_1_PROFIsafe_telegram_30"
      CU5_PN_1560A1_2_ModuleAccessPoint { ExternalAccessible := 'False'; ExternalVisible := 'False'; ExternalWritable := 'False'} : HW_SUBMODULE := 566;   // "CU5~PN~1560A1_2_ModuleAccessPoint"
      CU5_PN_1560A1_2_SIEMENS_telegram_111 { ExternalAccessible := 'False'; ExternalVisible := 'False'; ExternalWritable := 'False'} : HW_SUBMODULE := 567;   // "CU5~PN~1560A1_2_SIEMENS_telegram_111"
      CU5_PN_1560A1_2_PROFIsafe_telegram_30 { ExternalAccessible := 'False'; ExternalVisible := 'False'; ExternalWritable := 'False'} : HW_SUBMODULE := 568;   // "CU5~PN~1560A1_2_PROFIsafe_telegram_30"
      CU5_PN_1 { ExternalAccessible := 'False'; ExternalVisible := 'False'; ExternalWritable := 'False'} : HW_INTERFACE := 543;   // "CU5~PN(1)"
      CU5_PN_Port_1_1 { ExternalAccessible := 'False'; ExternalVisible := 'False'; ExternalWritable := 'False'} : HW_INTERFACE := 544;   // "CU5~PN~Port_1(1)"
      CU5_PN_Port_2_1 { ExternalAccessible := 'False'; ExternalVisible := 'False'; ExternalWritable := 'False'} : HW_INTERFACE := 545;   // "CU5~PN~Port_2(1)"
      CU5_PN_2 { ExternalAccessible := 'False'; ExternalVisible := 'False'; ExternalWritable := 'False'} : HW_INTERFACE := 543;   // "CU5~PN(2)"
      CU5_PN_Port_1_2 { ExternalAccessible := 'False'; ExternalVisible := 'False'; ExternalWritable := 'False'} : HW_INTERFACE := 544;   // "CU5~PN~Port_1(2)"
      CU5_PN_Port_2_2 { ExternalAccessible := 'False'; ExternalVisible := 'False'; ExternalWritable := 'False'} : HW_INTERFACE := 545;   // "CU5~PN~Port_2(2)"
      CU5_PN_3 { ExternalAccessible := 'False'; ExternalVisible := 'False'; ExternalWritable := 'False'} : HW_INTERFACE := 543;   // "CU5~PN(3)"
      CU5_PN_Port_1_3 { ExternalAccessible := 'False'; ExternalVisible := 'False'; ExternalWritable := 'False'} : HW_INTERFACE := 544;   // "CU5~PN~Port_1(3)"
      CU5_PN_Port_2_3 { ExternalAccessible := 'False'; ExternalVisible := 'False'; ExternalWritable := 'False'} : HW_INTERFACE := 545;   // "CU5~PN~Port_2(3)"
      CU6_PN_IODevice { ExternalAccessible := 'False'; ExternalVisible := 'False'; ExternalWritable := 'False'} : HW_DEVICE := 570;   // "CU6~PN~IODevice"
      CU6_PN { ExternalAccessible := 'False'; ExternalVisible := 'False'; ExternalWritable := 'False'} : HW_INTERFACE := 572;   // "CU6~PN"
      CU6_PN_Port_1 { ExternalAccessible := 'False'; ExternalVisible := 'False'; ExternalWritable := 'False'} : HW_INTERFACE := 573;   // "CU6~PN~Port_1"
      CU6_PN_Port_2 { ExternalAccessible := 'False'; ExternalVisible := 'False'; ExternalWritable := 'False'} : HW_INTERFACE := 574;   // "CU6~PN~Port_2"
      CU6_PN_605A1_ModuleAccessPoint { ExternalAccessible := 'False'; ExternalVisible := 'False'; ExternalWritable := 'False'} : HW_SUBMODULE := 576;   // "CU6~PN~605A1_ModuleAccessPoint"
      CU6_PN_605A1_SIEMENS_telegram_393 { ExternalAccessible := 'False'; ExternalVisible := 'False'; ExternalWritable := 'False'} : HW_SUBMODULE := 577;   // "CU6~PN~605A1_SIEMENS_telegram_393"
      CU6_PN_1990A1_1_ModuleAccessPoint { ExternalAccessible := 'False'; ExternalVisible := 'False'; ExternalWritable := 'False'} : HW_SUBMODULE := 579;   // "CU6~PN~1990A1_1_ModuleAccessPoint"
      CU6_PN_1990A1_1_PROFIsafe_telegram_30 { ExternalAccessible := 'False'; ExternalVisible := 'False'; ExternalWritable := 'False'} : HW_SUBMODULE := 581;   // "CU6~PN~1990A1_1_PROFIsafe_telegram_30"
      CU6_PN_1990A1_2_ModuleAccessPoint { ExternalAccessible := 'False'; ExternalVisible := 'False'; ExternalWritable := 'False'} : HW_SUBMODULE := 583;   // "CU6~PN~1990A1_2_ModuleAccessPoint"
      CU6_PN_1990A1_2_PROFIsafe_telegram_30 { ExternalAccessible := 'False'; ExternalVisible := 'False'; ExternalWritable := 'False'} : HW_SUBMODULE := 585;   // "CU6~PN~1990A1_2_PROFIsafe_telegram_30"
      CU6_PN_2100A1_1_ModuleAccessPoint { ExternalAccessible := 'False'; ExternalVisible := 'False'; ExternalWritable := 'False'} : HW_SUBMODULE := 587;   // "CU6~PN~2100A1_1_ModuleAccessPoint"
      CU6_PN_2100A1_1_SIEMENS_telegram_1 { ExternalAccessible := 'False'; ExternalVisible := 'False'; ExternalWritable := 'False'} : HW_SUBMODULE := 588;   // "CU6~PN~2100A1_1_SIEMENS_telegram_111"
      CU6_PN_2100A1_1_PROFIsafe_telegram_30 { ExternalAccessible := 'False'; ExternalVisible := 'False'; ExternalWritable := 'False'} : HW_SUBMODULE := 589;   // "CU6~PN~2100A1_1_PROFIsafe_telegram_30"
      CU6_PN_2100A1_2_ModuleAccessPoint { ExternalAccessible := 'False'; ExternalVisible := 'False'; ExternalWritable := 'False'} : HW_SUBMODULE := 591;   // "CU6~PN~2100A1_2_ModuleAccessPoint"
      CU6_PN_2100A1_2_SIEMENS_telegram_1 { ExternalAccessible := 'False'; ExternalVisible := 'False'; ExternalWritable := 'False'} : HW_SUBMODULE := 592;   // "CU6~PN~2100A1_2_SIEMENS_telegram_111"
      CU6_PN_2100A1_2_PROFIsafe_telegram_30 { ExternalAccessible := 'False'; ExternalVisible := 'False'; ExternalWritable := 'False'} : HW_SUBMODULE := 593;   // "CU6~PN~2100A1_2_PROFIsafe_telegram_30"
      CU6_PN_1840A1_1_ModuleAccessPoint { ExternalAccessible := 'False'; ExternalVisible := 'False'; ExternalWritable := 'False'} : HW_SUBMODULE := 599;   // "CU6~PN~1840A1_1_ModuleAccessPoint"
      CU6_PN_1840A1_1_PROFIsafe_telegram_30 { ExternalAccessible := 'False'; ExternalVisible := 'False'; ExternalWritable := 'False'} : HW_SUBMODULE := 601;   // "CU6~PN~1840A1_1_PROFIsafe_telegram_30"
      CU6_PN_1840A1_2_ModuleAccessPoint { ExternalAccessible := 'False'; ExternalVisible := 'False'; ExternalWritable := 'False'} : HW_SUBMODULE := 603;   // "CU6~PN~1840A1_2_ModuleAccessPoint"
      CU6_PN_1840A1_2_PROFIsafe_telegram_30 { ExternalAccessible := 'False'; ExternalVisible := 'False'; ExternalWritable := 'False'} : HW_SUBMODULE := 605;   // "CU6~PN~1840A1_2_PROFIsafe_telegram_30"
      CU6_PN_1 { ExternalAccessible := 'False'; ExternalVisible := 'False'; ExternalWritable := 'False'} : HW_INTERFACE := 572;   // "CU6~PN(1)"
      CU6_PN_Port_1_1 { ExternalAccessible := 'False'; ExternalVisible := 'False'; ExternalWritable := 'False'} : HW_INTERFACE := 573;   // "CU6~PN~Port_1(1)"
      CU6_PN_Port_2_1 { ExternalAccessible := 'False'; ExternalVisible := 'False'; ExternalWritable := 'False'} : HW_INTERFACE := 574;   // "CU6~PN~Port_2(1)"
      CU6_PN_2 { ExternalAccessible := 'False'; ExternalVisible := 'False'; ExternalWritable := 'False'} : HW_INTERFACE := 572;   // "CU6~PN(2)"
      CU6_PN_Port_1_2 { ExternalAccessible := 'False'; ExternalVisible := 'False'; ExternalWritable := 'False'} : HW_INTERFACE := 573;   // "CU6~PN~Port_1(2)"
      CU6_PN_Port_2_2 { ExternalAccessible := 'False'; ExternalVisible := 'False'; ExternalWritable := 'False'} : HW_INTERFACE := 574;   // "CU6~PN~Port_2(2)"
      CU6_PN_3 { ExternalAccessible := 'False'; ExternalVisible := 'False'; ExternalWritable := 'False'} : HW_INTERFACE := 572;   // "CU6~PN(3)"
      CU6_PN_Port_1_3 { ExternalAccessible := 'False'; ExternalVisible := 'False'; ExternalWritable := 'False'} : HW_INTERFACE := 573;   // "CU6~PN~Port_1(3)"
      CU6_PN_Port_2_3 { ExternalAccessible := 'False'; ExternalVisible := 'False'; ExternalWritable := 'False'} : HW_INTERFACE := 574;   // "CU6~PN~Port_2(3)"
      CU7_PN_IODevice { ExternalAccessible := 'False'; ExternalVisible := 'False'; ExternalWritable := 'False'} : HW_DEVICE := 607;   // "CU7~PN~IODevice"
      CU7_PN { ExternalAccessible := 'False'; ExternalVisible := 'False'; ExternalWritable := 'False'} : HW_INTERFACE := 609;   // "CU7~PN"
      CU7_PN_Port_1 { ExternalAccessible := 'False'; ExternalVisible := 'False'; ExternalWritable := 'False'} : HW_INTERFACE := 610;   // "CU7~PN~Port_1"
      CU7_PN_Port_2 { ExternalAccessible := 'False'; ExternalVisible := 'False'; ExternalWritable := 'False'} : HW_INTERFACE := 611;   // "CU7~PN~Port_2"
      CU7_PN_610A1_ModuleAccessPoint { ExternalAccessible := 'False'; ExternalVisible := 'False'; ExternalWritable := 'False'} : HW_SUBMODULE := 613;   // "CU7~PN~610A1_ModuleAccessPoint"
      CU7_PN_610A1_SIEMENS_telegram_393 { ExternalAccessible := 'False'; ExternalVisible := 'False'; ExternalWritable := 'False'} : HW_SUBMODULE := 614;   // "CU7~PN~610A1_SIEMENS_telegram_393"
      CU7_PN_2310A1_1_ModuleAccessPoint { ExternalAccessible := 'False'; ExternalVisible := 'False'; ExternalWritable := 'False'} : HW_SUBMODULE := 616;   // "CU7~PN~2310A1_1_ModuleAccessPoint"
      CU7_PN_2310A1_1_SIEMENS_telegram_111 { ExternalAccessible := 'False'; ExternalVisible := 'False'; ExternalWritable := 'False'} : HW_SUBMODULE := 617;   // "CU7~PN~2310A1_1_SIEMENS_telegram_111"
      CU7_PN_2310A1_1_PROFIsafe_telegram_30 { ExternalAccessible := 'False'; ExternalVisible := 'False'; ExternalWritable := 'False'} : HW_SUBMODULE := 618;   // "CU7~PN~2310A1_1_PROFIsafe_telegram_30"
      CU7_PN_2310A1_2_ModuleAccessPoint { ExternalAccessible := 'False'; ExternalVisible := 'False'; ExternalWritable := 'False'} : HW_SUBMODULE := 620;   // "CU7~PN~2310A1_2_ModuleAccessPoint"
      CU7_PN_2310A1_2_SIEMENS_telegram_111 { ExternalAccessible := 'False'; ExternalVisible := 'False'; ExternalWritable := 'False'} : HW_SUBMODULE := 621;   // "CU7~PN~2310A1_2_SIEMENS_telegram_111"
      CU7_PN_2310A1_2_PROFIsafe_telegram_30 { ExternalAccessible := 'False'; ExternalVisible := 'False'; ExternalWritable := 'False'} : HW_SUBMODULE := 622;   // "CU7~PN~2310A1_2_PROFIsafe_telegram_30"
      CU7_PN_2260A1_1_ModuleAccessPoint { ExternalAccessible := 'False'; ExternalVisible := 'False'; ExternalWritable := 'False'} : HW_SUBMODULE := 624;   // "CU7~PN~2260A1_1_ModuleAccessPoint"
      CU7_PN_2260A1_1_PROFIsafe_telegram_30 { ExternalAccessible := 'False'; ExternalVisible := 'False'; ExternalWritable := 'False'} : HW_SUBMODULE := 626;   // "CU7~PN~2260A1_1_PROFIsafe_telegram_30"
      CU7_PN_2260A1_2_ModuleAccessPoint { ExternalAccessible := 'False'; ExternalVisible := 'False'; ExternalWritable := 'False'} : HW_SUBMODULE := 628;   // "CU7~PN~2260A1_2_ModuleAccessPoint"
      CU7_PN_2260A1_2_PROFIsafe_telegram_30 { ExternalAccessible := 'False'; ExternalVisible := 'False'; ExternalWritable := 'False'} : HW_SUBMODULE := 630;   // "CU7~PN~2260A1_2_PROFIsafe_telegram_30"
      CU7_PN_2140A1_1_ModuleAccessPoint { ExternalAccessible := 'False'; ExternalVisible := 'False'; ExternalWritable := 'False'} : HW_SUBMODULE := 632;   // "CU7~PN~2140A1_1_ModuleAccessPoint"
      CU7_PN_2140A1_1_SIEMENS_telegram_111 { ExternalAccessible := 'False'; ExternalVisible := 'False'; ExternalWritable := 'False'} : HW_SUBMODULE := 633;   // "CU7~PN~2140A1_1_SIEMENS_telegram_111"
      CU7_PN_2140A1_1_PROFIsafe_telegram_30 { ExternalAccessible := 'False'; ExternalVisible := 'False'; ExternalWritable := 'False'} : HW_SUBMODULE := 634;   // "CU7~PN~2140A1_1_PROFIsafe_telegram_30"
      CU7_PN_2140A1_2_ModuleAccessPoint { ExternalAccessible := 'False'; ExternalVisible := 'False'; ExternalWritable := 'False'} : HW_SUBMODULE := 636;   // "CU7~PN~2140A1_2_ModuleAccessPoint"
      CU7_PN_2140A1_2_SIEMENS_telegram_111 { ExternalAccessible := 'False'; ExternalVisible := 'False'; ExternalWritable := 'False'} : HW_SUBMODULE := 637;   // "CU7~PN~2140A1_2_SIEMENS_telegram_111"
      CU7_PN_2140A1_2_PROFIsafe_telegram_30 { ExternalAccessible := 'False'; ExternalVisible := 'False'; ExternalWritable := 'False'} : HW_SUBMODULE := 638;   // "CU7~PN~2140A1_2_PROFIsafe_telegram_30"
      CU7_PN_1 { ExternalAccessible := 'False'; ExternalVisible := 'False'; ExternalWritable := 'False'} : HW_INTERFACE := 609;   // "CU7~PN(1)"
      CU7_PN_Port_1_1 { ExternalAccessible := 'False'; ExternalVisible := 'False'; ExternalWritable := 'False'} : HW_INTERFACE := 610;   // "CU7~PN~Port_1(1)"
      CU7_PN_Port_2_1 { ExternalAccessible := 'False'; ExternalVisible := 'False'; ExternalWritable := 'False'} : HW_INTERFACE := 611;   // "CU7~PN~Port_2(1)"
      CU7_PN_2 { ExternalAccessible := 'False'; ExternalVisible := 'False'; ExternalWritable := 'False'} : HW_INTERFACE := 609;   // "CU7~PN(2)"
      CU7_PN_Port_1_2 { ExternalAccessible := 'False'; ExternalVisible := 'False'; ExternalWritable := 'False'} : HW_INTERFACE := 610;   // "CU7~PN~Port_1(2)"
      CU7_PN_Port_2_2 { ExternalAccessible := 'False'; ExternalVisible := 'False'; ExternalWritable := 'False'} : HW_INTERFACE := 611;   // "CU7~PN~Port_2(2)"
      CU7_PN_3 { ExternalAccessible := 'False'; ExternalVisible := 'False'; ExternalWritable := 'False'} : HW_INTERFACE := 609;   // "CU7~PN(3)"
      CU7_PN_Port_1_3 { ExternalAccessible := 'False'; ExternalVisible := 'False'; ExternalWritable := 'False'} : HW_INTERFACE := 610;   // "CU7~PN~Port_1(3)"
      CU7_PN_Port_2_3 { ExternalAccessible := 'False'; ExternalVisible := 'False'; ExternalWritable := 'False'} : HW_INTERFACE := 611;   // "CU7~PN~Port_2(3)"
      CU8_PN_IODevice { ExternalAccessible := 'False'; ExternalVisible := 'False'; ExternalWritable := 'False'} : HW_DEVICE := 640;   // "CU8~PN~IODevice"
      CU8_PN { ExternalAccessible := 'False'; ExternalVisible := 'False'; ExternalWritable := 'False'} : HW_INTERFACE := 642;   // "CU8~PN"
      CU8_PN_Port_1 { ExternalAccessible := 'False'; ExternalVisible := 'False'; ExternalWritable := 'False'} : HW_INTERFACE := 643;   // "CU8~PN~Port_1"
      CU8_PN_Port_2 { ExternalAccessible := 'False'; ExternalVisible := 'False'; ExternalWritable := 'False'} : HW_INTERFACE := 644;   // "CU8~PN~Port_2"
      CU8_PN_615A1_ModuleAccessPoint { ExternalAccessible := 'False'; ExternalVisible := 'False'; ExternalWritable := 'False'} : HW_SUBMODULE := 646;   // "CU8~PN~615A1_ModuleAccessPoint"
      CU8_PN_615A1_SIEMENS_telegram_393 { ExternalAccessible := 'False'; ExternalVisible := 'False'; ExternalWritable := 'False'} : HW_SUBMODULE := 647;   // "CU8~PN~615A1_SIEMENS_telegram_393"
      CU8_PN_2390A1_1_ModuleAccessPoint { ExternalAccessible := 'False'; ExternalVisible := 'False'; ExternalWritable := 'False'} : HW_SUBMODULE := 649;   // "CU8~PN~2390A1_1_ModuleAccessPoint"
      CU8_PN_2390A1_1_PROFIsafe_telegram_30 { ExternalAccessible := 'False'; ExternalVisible := 'False'; ExternalWritable := 'False'} : HW_SUBMODULE := 650;   // "CU8~PN~2390A1_1_PROFIsafe_telegram_30"
      CU8_PN_2390A1_2_ModuleAccessPoint { ExternalAccessible := 'False'; ExternalVisible := 'False'; ExternalWritable := 'False'} : HW_SUBMODULE := 653;   // "CU8~PN~2390A1_2_ModuleAccessPoint"
      CU8_PN_2390A1_2_PROFIsafe_telegram_30 { ExternalAccessible := 'False'; ExternalVisible := 'False'; ExternalWritable := 'False'} : HW_SUBMODULE := 654;   // "CU8~PN~2390A1_2_PROFIsafe_telegram_30"
      CU8_PN_2430A1_1_ModuleAccessPoint { ExternalAccessible := 'False'; ExternalVisible := 'False'; ExternalWritable := 'False'} : HW_SUBMODULE := 657;   // "CU8~PN~2430A1_1_ModuleAccessPoint"
      CU8_PN_2430A1_1_PROFIsafe_telegram_30 { ExternalAccessible := 'False'; ExternalVisible := 'False'; ExternalWritable := 'False'} : HW_SUBMODULE := 658;   // "CU8~PN~2430A1_1_PROFIsafe_telegram_30"
      CU8_PN_2430A1_2_ModuleAccessPoint { ExternalAccessible := 'False'; ExternalVisible := 'False'; ExternalWritable := 'False'} : HW_SUBMODULE := 661;   // "CU8~PN~2430A1_2_ModuleAccessPoint"
      CU8_PN_2430A1_2_PROFIsafe_telegram_30 { ExternalAccessible := 'False'; ExternalVisible := 'False'; ExternalWritable := 'False'} : HW_SUBMODULE := 662;   // "CU8~PN~2430A1_2_PROFIsafe_telegram_30"
      CU8_PN_2350A1_1_ModuleAccessPoint { ExternalAccessible := 'False'; ExternalVisible := 'False'; ExternalWritable := 'False'} : HW_SUBMODULE := 665;   // "CU8~PN~2350A1_1_ModuleAccessPoint"
      CU8_PN_2350A1_1_PROFIsafe_telegram_30 { ExternalAccessible := 'False'; ExternalVisible := 'False'; ExternalWritable := 'False'} : HW_SUBMODULE := 666;   // "CU8~PN~2350A1_1_PROFIsafe_telegram_30"
      CU8_PN_2350A1_2_ModuleAccessPoint { ExternalAccessible := 'False'; ExternalVisible := 'False'; ExternalWritable := 'False'} : HW_SUBMODULE := 669;   // "CU8~PN~2350A1_2_ModuleAccessPoint"
      CU8_PN_2350A1_2_PROFIsafe_telegram_30 { ExternalAccessible := 'False'; ExternalVisible := 'False'; ExternalWritable := 'False'} : HW_SUBMODULE := 670;   // "CU8~PN~2350A1_2_PROFIsafe_telegram_30"
      CU8_PN_640A1_ModuleAccessPoint { ExternalAccessible := 'False'; ExternalVisible := 'False'; ExternalWritable := 'False'} : HW_SUBMODULE := 673;   // "CU8~PN~640A1_ModuleAccessPoint"
      CU8_PN_640A1_SIEMENS_telegram_370 { ExternalAccessible := 'False'; ExternalVisible := 'False'; ExternalWritable := 'False'} : HW_SUBMODULE := 674;   // "CU8~PN~640A1_SIEMENS_telegram_370"
      CU8_PN_1 { ExternalAccessible := 'False'; ExternalVisible := 'False'; ExternalWritable := 'False'} : HW_INTERFACE := 642;   // "CU8~PN(1)"
      CU8_PN_Port_1_1 { ExternalAccessible := 'False'; ExternalVisible := 'False'; ExternalWritable := 'False'} : HW_INTERFACE := 643;   // "CU8~PN~Port_1(1)"
      CU8_PN_Port_2_1 { ExternalAccessible := 'False'; ExternalVisible := 'False'; ExternalWritable := 'False'} : HW_INTERFACE := 644;   // "CU8~PN~Port_2(1)"
      CU8_PN_2 { ExternalAccessible := 'False'; ExternalVisible := 'False'; ExternalWritable := 'False'} : HW_INTERFACE := 642;   // "CU8~PN(2)"
      CU8_PN_Port_1_2 { ExternalAccessible := 'False'; ExternalVisible := 'False'; ExternalWritable := 'False'} : HW_INTERFACE := 643;   // "CU8~PN~Port_1(2)"
      CU8_PN_Port_2_2 { ExternalAccessible := 'False'; ExternalVisible := 'False'; ExternalWritable := 'False'} : HW_INTERFACE := 644;   // "CU8~PN~Port_2(2)"
      CU8_PN_3 { ExternalAccessible := 'False'; ExternalVisible := 'False'; ExternalWritable := 'False'} : HW_INTERFACE := 642;   // "CU8~PN(3)"
      CU8_PN_Port_1_3 { ExternalAccessible := 'False'; ExternalVisible := 'False'; ExternalWritable := 'False'} : HW_INTERFACE := 643;   // "CU8~PN~Port_1(3)"
      CU8_PN_Port_2_3 { ExternalAccessible := 'False'; ExternalVisible := 'False'; ExternalWritable := 'False'} : HW_INTERFACE := 644;   // "CU8~PN~Port_2(3)"
      HW_1008P1_Proxy { ExternalAccessible := 'False'; ExternalVisible := 'False'; ExternalWritable := 'False'} : HW_SUBMODULE := 684;   // "1008P1~Proxy"
      HW_1008P1_IODevice { ExternalAccessible := 'False'; ExternalVisible := 'False'; ExternalWritable := 'False'} : HW_DEVICE := 682;   // "1008P1~IODevice"
      HW_1008P1_Interface { ExternalAccessible := 'False'; ExternalVisible := 'False'; ExternalWritable := 'False'} : HW_INTERFACE := 685;   // "1008P1~Interface"
      HW_1008P1_Interface_Port_1 { ExternalAccessible := 'False'; ExternalVisible := 'False'; ExternalWritable := 'False'} : HW_INTERFACE := 686;   // "1008P1~Interface~Port_1"
      HW_1008P1_Interface_Port_2 { ExternalAccessible := 'False'; ExternalVisible := 'False'; ExternalWritable := 'False'} : HW_INTERFACE := 687;   // "1008P1~Interface~Port_2"
      HW_1008P1_Head { ExternalAccessible := 'False'; ExternalVisible := 'False'; ExternalWritable := 'False'} : HW_SUBMODULE := 688;   // "1008P1~Head"
      HW_1008P1_EO_Multiturn_1 { ExternalAccessible := 'False'; ExternalVisible := 'False'; ExternalWritable := 'False'} : HW_SUBMODULE := 689;   // "1008P1~EO_Multiturn_1"
      HW_1008P1_Telegram_81_DI_DO { ExternalAccessible := 'False'; ExternalVisible := 'False'; ExternalWritable := 'False'} : HW_SUBMODULE := 690;   // "1008P1_Telegram_81~DI_DO"
      HW_1008P1_EO_Multiturn_1_Parameter_Access_Point { ExternalAccessible := 'False'; ExternalVisible := 'False'; ExternalWritable := 'False'} : HW_SUBMODULE := 691;   // "1008P1~EO_Multiturn_1~Parameter_Access_Point"
      HW_1004P1_Proxy { ExternalAccessible := 'False'; ExternalVisible := 'False'; ExternalWritable := 'False'} : HW_SUBMODULE := 694;   // "1004P1~Proxy"
      HW_1004P1_IODevice { ExternalAccessible := 'False'; ExternalVisible := 'False'; ExternalWritable := 'False'} : HW_DEVICE := 692;   // "1004P1~IODevice"
      HW_1004P1_Interface { ExternalAccessible := 'False'; ExternalVisible := 'False'; ExternalWritable := 'False'} : HW_INTERFACE := 695;   // "1004P1~Interface"
      HW_1004P1_Interface_Port_1 { ExternalAccessible := 'False'; ExternalVisible := 'False'; ExternalWritable := 'False'} : HW_INTERFACE := 696;   // "1004P1~Interface~Port_1"
      HW_1004P1_Interface_Port_2 { ExternalAccessible := 'False'; ExternalVisible := 'False'; ExternalWritable := 'False'} : HW_INTERFACE := 697;   // "1004P1~Interface~Port_2"
      HW_1004P1_Head { ExternalAccessible := 'False'; ExternalVisible := 'False'; ExternalWritable := 'False'} : HW_SUBMODULE := 698;   // "1004P1~Head"
      HW_1004P1_EO_Multiturn_1 { ExternalAccessible := 'False'; ExternalVisible := 'False'; ExternalWritable := 'False'} : HW_SUBMODULE := 699;   // "1004P1~EO_Multiturn_1"
      HW_1004P1_Telegram_81_DI_DO { ExternalAccessible := 'False'; ExternalVisible := 'False'; ExternalWritable := 'False'} : HW_SUBMODULE := 700;   // "1004P1_Telegram_81~DI_DO"
      HW_1004P1_EO_Multiturn_1_Parameter_Access_Point { ExternalAccessible := 'False'; ExternalVisible := 'False'; ExternalWritable := 'False'} : HW_SUBMODULE := 701;   // "1004P1~EO_Multiturn_1~Parameter_Access_Point"
      HW_994P1_Proxy { ExternalAccessible := 'False'; ExternalVisible := 'False'; ExternalWritable := 'False'} : HW_SUBMODULE := 726;   // "994P1~Proxy"
      HW_994P1_IODevice { ExternalAccessible := 'False'; ExternalVisible := 'False'; ExternalWritable := 'False'} : HW_DEVICE := 724;   // "994P1~IODevice"
      HW_994P1_Interface { ExternalAccessible := 'False'; ExternalVisible := 'False'; ExternalWritable := 'False'} : HW_INTERFACE := 727;   // "994P1~Interface"
      HW_994P1_Interface_Port_1 { ExternalAccessible := 'False'; ExternalVisible := 'False'; ExternalWritable := 'False'} : HW_INTERFACE := 728;   // "994P1~Interface~Port_1"
      HW_994P1_Interface_Port_2 { ExternalAccessible := 'False'; ExternalVisible := 'False'; ExternalWritable := 'False'} : HW_INTERFACE := 729;   // "994P1~Interface~Port_2"
      HW_994P1_Head { ExternalAccessible := 'False'; ExternalVisible := 'False'; ExternalWritable := 'False'} : HW_SUBMODULE := 730;   // "994P1~Head"
      HW_994P1_EO_Multiturn_1 { ExternalAccessible := 'False'; ExternalVisible := 'False'; ExternalWritable := 'False'} : HW_SUBMODULE := 731;   // "994P1~EO_Multiturn_1"
      HW_994P1_Telegram_81_DI_DO { ExternalAccessible := 'False'; ExternalVisible := 'False'; ExternalWritable := 'False'} : HW_SUBMODULE := 732;   // "994P1_Telegram_81~DI_DO"
      HW_994P1_EO_Multiturn_1_Parameter_Access_Point { ExternalAccessible := 'False'; ExternalVisible := 'False'; ExternalWritable := 'False'} : HW_SUBMODULE := 733;   // "994P1~EO_Multiturn_1~Parameter_Access_Point"
      HW_984P1_Proxy { ExternalAccessible := 'False'; ExternalVisible := 'False'; ExternalWritable := 'False'} : HW_SUBMODULE := 736;   // "984P1~Proxy"
      HW_984P1_IODevice { ExternalAccessible := 'False'; ExternalVisible := 'False'; ExternalWritable := 'False'} : HW_DEVICE := 734;   // "984P1~IODevice"
      HW_984P1_Interface { ExternalAccessible := 'False'; ExternalVisible := 'False'; ExternalWritable := 'False'} : HW_INTERFACE := 737;   // "984P1~Interface"
      HW_984P1_Interface_Port_1 { ExternalAccessible := 'False'; ExternalVisible := 'False'; ExternalWritable := 'False'} : HW_INTERFACE := 738;   // "984P1~Interface~Port_1"
      HW_984P1_Interface_Port_2 { ExternalAccessible := 'False'; ExternalVisible := 'False'; ExternalWritable := 'False'} : HW_INTERFACE := 739;   // "984P1~Interface~Port_2"
      HW_984P1_Head { ExternalAccessible := 'False'; ExternalVisible := 'False'; ExternalWritable := 'False'} : HW_SUBMODULE := 740;   // "984P1~Head"
      HW_984P1_EO_Multiturn_1 { ExternalAccessible := 'False'; ExternalVisible := 'False'; ExternalWritable := 'False'} : HW_SUBMODULE := 741;   // "984P1~EO_Multiturn_1"
      HW_984P1_Telegram_81_DI_DO { ExternalAccessible := 'False'; ExternalVisible := 'False'; ExternalWritable := 'False'} : HW_SUBMODULE := 742;   // "984P1_Telegram_81~DI_DO"
      HW_984P1_EO_Multiturn_1_Parameter_Access_Point { ExternalAccessible := 'False'; ExternalVisible := 'False'; ExternalWritable := 'False'} : HW_SUBMODULE := 743;   // "984P1~EO_Multiturn_1~Parameter_Access_Point"
      HW_1868P1_Proxy { ExternalAccessible := 'False'; ExternalVisible := 'False'; ExternalWritable := 'False'} : HW_SUBMODULE := 873;   // "1868P1~Proxy"
      HW_1868P1_IODevice { ExternalAccessible := 'False'; ExternalVisible := 'False'; ExternalWritable := 'False'} : HW_DEVICE := 871;   // "1868P1~IODevice"
      HW_1868P1_Interface { ExternalAccessible := 'False'; ExternalVisible := 'False'; ExternalWritable := 'False'} : HW_INTERFACE := 874;   // "1868P1~Interface"
      HW_1868P1_Interface_Port_1 { ExternalAccessible := 'False'; ExternalVisible := 'False'; ExternalWritable := 'False'} : HW_INTERFACE := 875;   // "1868P1~Interface~Port_1"
      HW_1868P1_Interface_Port_2 { ExternalAccessible := 'False'; ExternalVisible := 'False'; ExternalWritable := 'False'} : HW_INTERFACE := 876;   // "1868P1~Interface~Port_2"
      HW_1868P1_Head { ExternalAccessible := 'False'; ExternalVisible := 'False'; ExternalWritable := 'False'} : HW_SUBMODULE := 877;   // "1868P1~Head"
      HW_1868P1_EO_Multiturn_1 { ExternalAccessible := 'False'; ExternalVisible := 'False'; ExternalWritable := 'False'} : HW_SUBMODULE := 878;   // "1868P1~EO_Multiturn_1"
      HW_1868P1_Telegram_81_DI_DO { ExternalAccessible := 'False'; ExternalVisible := 'False'; ExternalWritable := 'False'} : HW_SUBMODULE := 879;   // "1868P1_Telegram_81~DI_DO"
      HW_1868P1_EO_Multiturn_1_Parameter_Access_Point { ExternalAccessible := 'False'; ExternalVisible := 'False'; ExternalWritable := 'False'} : HW_SUBMODULE := 880;   // "1868P1~EO_Multiturn_1~Parameter_Access_Point"
      HW_1863P1_Proxy { ExternalAccessible := 'False'; ExternalVisible := 'False'; ExternalWritable := 'False'} : HW_SUBMODULE := 883;   // "1863P1~Proxy"
      HW_1863P1_IODevice { ExternalAccessible := 'False'; ExternalVisible := 'False'; ExternalWritable := 'False'} : HW_DEVICE := 881;   // "1863P1~IODevice"
      HW_1863P1_Interface { ExternalAccessible := 'False'; ExternalVisible := 'False'; ExternalWritable := 'False'} : HW_INTERFACE := 884;   // "1863P1~Interface"
      HW_1863P1_Interface_Port_1 { ExternalAccessible := 'False'; ExternalVisible := 'False'; ExternalWritable := 'False'} : HW_INTERFACE := 885;   // "1863P1~Interface~Port_1"
      HW_1863P1_Interface_Port_2 { ExternalAccessible := 'False'; ExternalVisible := 'False'; ExternalWritable := 'False'} : HW_INTERFACE := 886;   // "1863P1~Interface~Port_2"
      HW_1863P1_Head { ExternalAccessible := 'False'; ExternalVisible := 'False'; ExternalWritable := 'False'} : HW_SUBMODULE := 887;   // "1863P1~Head"
      HW_1863P1_EO_Multiturn_1 { ExternalAccessible := 'False'; ExternalVisible := 'False'; ExternalWritable := 'False'} : HW_SUBMODULE := 888;   // "1863P1~EO_Multiturn_1"
      HW_1863P1_Telegram_81_DI_DO { ExternalAccessible := 'False'; ExternalVisible := 'False'; ExternalWritable := 'False'} : HW_SUBMODULE := 889;   // "1863P1_Telegram_81~DI_DO"
      HW_1863P1_EO_Multiturn_1_Parameter_Access_Point { ExternalAccessible := 'False'; ExternalVisible := 'False'; ExternalWritable := 'False'} : HW_SUBMODULE := 890;   // "1863P1~EO_Multiturn_1~Parameter_Access_Point"
      HW_1858P1_Proxy { ExternalAccessible := 'False'; ExternalVisible := 'False'; ExternalWritable := 'False'} : HW_SUBMODULE := 893;   // "1858P1~Proxy"
      HW_1858P1_IODevice { ExternalAccessible := 'False'; ExternalVisible := 'False'; ExternalWritable := 'False'} : HW_DEVICE := 891;   // "1858P1~IODevice"
      HW_1858P1_Interface { ExternalAccessible := 'False'; ExternalVisible := 'False'; ExternalWritable := 'False'} : HW_INTERFACE := 894;   // "1858P1~Interface"
      HW_1858P1_Interface_Port_1 { ExternalAccessible := 'False'; ExternalVisible := 'False'; ExternalWritable := 'False'} : HW_INTERFACE := 895;   // "1858P1~Interface~Port_1"
      HW_1858P1_Interface_Port_2 { ExternalAccessible := 'False'; ExternalVisible := 'False'; ExternalWritable := 'False'} : HW_INTERFACE := 896;   // "1858P1~Interface~Port_2"
      HW_1858P1_Head { ExternalAccessible := 'False'; ExternalVisible := 'False'; ExternalWritable := 'False'} : HW_SUBMODULE := 897;   // "1858P1~Head"
      HW_1858P1_EO_Multiturn_1 { ExternalAccessible := 'False'; ExternalVisible := 'False'; ExternalWritable := 'False'} : HW_SUBMODULE := 898;   // "1858P1~EO_Multiturn_1"
      HW_1858P1_Telegram_81_DI_DO { ExternalAccessible := 'False'; ExternalVisible := 'False'; ExternalWritable := 'False'} : HW_SUBMODULE := 899;   // "1858P1_Telegram_81~DI_DO"
      HW_1858P1_EO_Multiturn_1_Parameter_Access_Point { ExternalAccessible := 'False'; ExternalVisible := 'False'; ExternalWritable := 'False'} : HW_SUBMODULE := 900;   // "1858P1~EO_Multiturn_1~Parameter_Access_Point"
      HW_1853P1_Proxy { ExternalAccessible := 'False'; ExternalVisible := 'False'; ExternalWritable := 'False'} : HW_SUBMODULE := 903;   // "1853P1~Proxy"
      HW_1853P1_IODevice { ExternalAccessible := 'False'; ExternalVisible := 'False'; ExternalWritable := 'False'} : HW_DEVICE := 901;   // "1853P1~IODevice"
      HW_1853P1_Interface { ExternalAccessible := 'False'; ExternalVisible := 'False'; ExternalWritable := 'False'} : HW_INTERFACE := 904;   // "1853P1~Interface"
      HW_1853P1_Interface_Port_1 { ExternalAccessible := 'False'; ExternalVisible := 'False'; ExternalWritable := 'False'} : HW_INTERFACE := 905;   // "1853P1~Interface~Port_1"
      HW_1853P1_Interface_Port_2 { ExternalAccessible := 'False'; ExternalVisible := 'False'; ExternalWritable := 'False'} : HW_INTERFACE := 906;   // "1853P1~Interface~Port_2"
      HW_1853P1_Head { ExternalAccessible := 'False'; ExternalVisible := 'False'; ExternalWritable := 'False'} : HW_SUBMODULE := 907;   // "1853P1~Head"
      HW_1853P1_EO_Multiturn_1 { ExternalAccessible := 'False'; ExternalVisible := 'False'; ExternalWritable := 'False'} : HW_SUBMODULE := 908;   // "1853P1~EO_Multiturn_1"
      HW_1853P1_Telegram_81_DI_DO { ExternalAccessible := 'False'; ExternalVisible := 'False'; ExternalWritable := 'False'} : HW_SUBMODULE := 909;   // "1853P1_Telegram_81~DI_DO"
      HW_1853P1_EO_Multiturn_1_Parameter_Access_Point { ExternalAccessible := 'False'; ExternalVisible := 'False'; ExternalWritable := 'False'} : HW_SUBMODULE := 910;   // "1853P1~EO_Multiturn_1~Parameter_Access_Point"
      HW_1844P1_Proxy { ExternalAccessible := 'False'; ExternalVisible := 'False'; ExternalWritable := 'False'} : HW_SUBMODULE := 913;   // "1844P1~Proxy"
      HW_1844P1_IODevice { ExternalAccessible := 'False'; ExternalVisible := 'False'; ExternalWritable := 'False'} : HW_DEVICE := 911;   // "1844P1~IODevice"
      HW_1844P1_Interface { ExternalAccessible := 'False'; ExternalVisible := 'False'; ExternalWritable := 'False'} : HW_INTERFACE := 914;   // "1844P1~Interface"
      HW_1844P1_Interface_Port_1 { ExternalAccessible := 'False'; ExternalVisible := 'False'; ExternalWritable := 'False'} : HW_INTERFACE := 915;   // "1844P1~Interface~Port_1"
      HW_1844P1_Interface_Port_2 { ExternalAccessible := 'False'; ExternalVisible := 'False'; ExternalWritable := 'False'} : HW_INTERFACE := 916;   // "1844P1~Interface~Port_2"
      HW_1844P1_Head { ExternalAccessible := 'False'; ExternalVisible := 'False'; ExternalWritable := 'False'} : HW_SUBMODULE := 917;   // "1844P1~Head"
      HW_1844P1_EO_Multiturn_1 { ExternalAccessible := 'False'; ExternalVisible := 'False'; ExternalWritable := 'False'} : HW_SUBMODULE := 918;   // "1844P1~EO_Multiturn_1"
      HW_1844P1_Telegram_81_DI_DO { ExternalAccessible := 'False'; ExternalVisible := 'False'; ExternalWritable := 'False'} : HW_SUBMODULE := 919;   // "1844P1_Telegram_81~DI_DO"
      HW_1844P1_EO_Multiturn_1_Parameter_Access_Point { ExternalAccessible := 'False'; ExternalVisible := 'False'; ExternalWritable := 'False'} : HW_SUBMODULE := 920;   // "1844P1~EO_Multiturn_1~Parameter_Access_Point"
      HW_1044P1_Proxy { ExternalAccessible := 'False'; ExternalVisible := 'False'; ExternalWritable := 'False'} : HW_SUBMODULE := 746;   // "1044P1~Proxy"
      HW_1044P1_IODevice { ExternalAccessible := 'False'; ExternalVisible := 'False'; ExternalWritable := 'False'} : HW_DEVICE := 744;   // "1044P1~IODevice"
      HW_1044P1_Interface { ExternalAccessible := 'False'; ExternalVisible := 'False'; ExternalWritable := 'False'} : HW_INTERFACE := 747;   // "1044P1~Interface"
      HW_1044P1_Interface_Port_1 { ExternalAccessible := 'False'; ExternalVisible := 'False'; ExternalWritable := 'False'} : HW_INTERFACE := 748;   // "1044P1~Interface~Port_1"
      HW_1044P1_Interface_Port_2 { ExternalAccessible := 'False'; ExternalVisible := 'False'; ExternalWritable := 'False'} : HW_INTERFACE := 749;   // "1044P1~Interface~Port_2"
      HW_1044P1_Head { ExternalAccessible := 'False'; ExternalVisible := 'False'; ExternalWritable := 'False'} : HW_SUBMODULE := 750;   // "1044P1~Head"
      HW_1044P1_EO_Multiturn_1 { ExternalAccessible := 'False'; ExternalVisible := 'False'; ExternalWritable := 'False'} : HW_SUBMODULE := 751;   // "1044P1~EO_Multiturn_1"
      HW_1044P1_Telegram_81_DI_DO { ExternalAccessible := 'False'; ExternalVisible := 'False'; ExternalWritable := 'False'} : HW_SUBMODULE := 752;   // "1044P1_Telegram_81~DI_DO"
      HW_1044P1_EO_Multiturn_1_Parameter_Access_Point { ExternalAccessible := 'False'; ExternalVisible := 'False'; ExternalWritable := 'False'} : HW_SUBMODULE := 753;   // "1044P1~EO_Multiturn_1~Parameter_Access_Point"
      HW_1034P1_Proxy { ExternalAccessible := 'False'; ExternalVisible := 'False'; ExternalWritable := 'False'} : HW_SUBMODULE := 756;   // "1034P1~Proxy"
      HW_1034P1_IODevice { ExternalAccessible := 'False'; ExternalVisible := 'False'; ExternalWritable := 'False'} : HW_DEVICE := 754;   // "1034P1~IODevice"
      HW_1034P1_Interface { ExternalAccessible := 'False'; ExternalVisible := 'False'; ExternalWritable := 'False'} : HW_INTERFACE := 757;   // "1034P1~Interface"
      HW_1034P1_Interface_Port_1 { ExternalAccessible := 'False'; ExternalVisible := 'False'; ExternalWritable := 'False'} : HW_INTERFACE := 758;   // "1034P1~Interface~Port_1"
      HW_1034P1_Interface_Port_2 { ExternalAccessible := 'False'; ExternalVisible := 'False'; ExternalWritable := 'False'} : HW_INTERFACE := 759;   // "1034P1~Interface~Port_2"
      HW_1034P1_Head { ExternalAccessible := 'False'; ExternalVisible := 'False'; ExternalWritable := 'False'} : HW_SUBMODULE := 760;   // "1034P1~Head"
      HW_1034P1_EO_Multiturn_1 { ExternalAccessible := 'False'; ExternalVisible := 'False'; ExternalWritable := 'False'} : HW_SUBMODULE := 761;   // "1034P1~EO_Multiturn_1"
      HW_1034P1_Telegram_81_DI_DO { ExternalAccessible := 'False'; ExternalVisible := 'False'; ExternalWritable := 'False'} : HW_SUBMODULE := 762;   // "1034P1_Telegram_81~DI_DO"
      HW_1034P1_EO_Multiturn_1_Parameter_Access_Point { ExternalAccessible := 'False'; ExternalVisible := 'False'; ExternalWritable := 'False'} : HW_SUBMODULE := 763;   // "1034P1~EO_Multiturn_1~Parameter_Access_Point"
      HW_1918P1_Proxy { ExternalAccessible := 'False'; ExternalVisible := 'False'; ExternalWritable := 'False'} : HW_SUBMODULE := 923;   // "1918P1~Proxy"
      HW_1918P1_IODevice { ExternalAccessible := 'False'; ExternalVisible := 'False'; ExternalWritable := 'False'} : HW_DEVICE := 921;   // "1918P1~IODevice"
      HW_1918P1_Interface { ExternalAccessible := 'False'; ExternalVisible := 'False'; ExternalWritable := 'False'} : HW_INTERFACE := 924;   // "1918P1~Interface"
      HW_1918P1_Interface_Port_1 { ExternalAccessible := 'False'; ExternalVisible := 'False'; ExternalWritable := 'False'} : HW_INTERFACE := 925;   // "1918P1~Interface~Port_1"
      HW_1918P1_Interface_Port_2 { ExternalAccessible := 'False'; ExternalVisible := 'False'; ExternalWritable := 'False'} : HW_INTERFACE := 926;   // "1918P1~Interface~Port_2"
      HW_1918P1_Head { ExternalAccessible := 'False'; ExternalVisible := 'False'; ExternalWritable := 'False'} : HW_SUBMODULE := 927;   // "1918P1~Head"
      HW_1918P1_EO_Multiturn_1 { ExternalAccessible := 'False'; ExternalVisible := 'False'; ExternalWritable := 'False'} : HW_SUBMODULE := 928;   // "1918P1~EO_Multiturn_1"
      HW_1918P1_Telegram_81_DI_DO { ExternalAccessible := 'False'; ExternalVisible := 'False'; ExternalWritable := 'False'} : HW_SUBMODULE := 929;   // "1918P1_Telegram_81~DI_DO"
      HW_1918P1_EO_Multiturn_1_Parameter_Access_Point { ExternalAccessible := 'False'; ExternalVisible := 'False'; ExternalWritable := 'False'} : HW_SUBMODULE := 930;   // "1918P1~EO_Multiturn_1~Parameter_Access_Point"
      HW_1093P1_Proxy { ExternalAccessible := 'False'; ExternalVisible := 'False'; ExternalWritable := 'False'} : HW_SUBMODULE := 766;   // "1093P1~Proxy"
      HW_1093P1_IODevice { ExternalAccessible := 'False'; ExternalVisible := 'False'; ExternalWritable := 'False'} : HW_DEVICE := 764;   // "1093P1~IODevice"
      HW_1093P1_Interface { ExternalAccessible := 'False'; ExternalVisible := 'False'; ExternalWritable := 'False'} : HW_INTERFACE := 767;   // "1093P1~Interface"
      HW_1093P1_Interface_Port_1 { ExternalAccessible := 'False'; ExternalVisible := 'False'; ExternalWritable := 'False'} : HW_INTERFACE := 768;   // "1093P1~Interface~Port_1"
      HW_1093P1_Interface_Port_2 { ExternalAccessible := 'False'; ExternalVisible := 'False'; ExternalWritable := 'False'} : HW_INTERFACE := 769;   // "1093P1~Interface~Port_2"
      HW_1093P1_Head { ExternalAccessible := 'False'; ExternalVisible := 'False'; ExternalWritable := 'False'} : HW_SUBMODULE := 770;   // "1093P1~Head"
      HW_1093P1_EO_Multiturn_1 { ExternalAccessible := 'False'; ExternalVisible := 'False'; ExternalWritable := 'False'} : HW_SUBMODULE := 771;   // "1093P1~EO_Multiturn_1"
      HW_1093P1_Telegram_81_DI_DO { ExternalAccessible := 'False'; ExternalVisible := 'False'; ExternalWritable := 'False'} : HW_SUBMODULE := 772;   // "1093P1_Telegram_81~DI_DO"
      HW_1093P1_EO_Multiturn_1_Parameter_Access_Point { ExternalAccessible := 'False'; ExternalVisible := 'False'; ExternalWritable := 'False'} : HW_SUBMODULE := 773;   // "1093P1~EO_Multiturn_1~Parameter_Access_Point"
      HW_1913P1_Proxy { ExternalAccessible := 'False'; ExternalVisible := 'False'; ExternalWritable := 'False'} : HW_SUBMODULE := 933;   // "1913P1~Proxy"
      HW_1913P1_IODevice { ExternalAccessible := 'False'; ExternalVisible := 'False'; ExternalWritable := 'False'} : HW_DEVICE := 931;   // "1913P1~IODevice"
      HW_1913P1_Interface { ExternalAccessible := 'False'; ExternalVisible := 'False'; ExternalWritable := 'False'} : HW_INTERFACE := 934;   // "1913P1~Interface"
      HW_1913P1_Interface_Port_1 { ExternalAccessible := 'False'; ExternalVisible := 'False'; ExternalWritable := 'False'} : HW_INTERFACE := 935;   // "1913P1~Interface~Port_1"
      HW_1913P1_Interface_Port_2 { ExternalAccessible := 'False'; ExternalVisible := 'False'; ExternalWritable := 'False'} : HW_INTERFACE := 936;   // "1913P1~Interface~Port_2"
      HW_1913P1_Head { ExternalAccessible := 'False'; ExternalVisible := 'False'; ExternalWritable := 'False'} : HW_SUBMODULE := 937;   // "1913P1~Head"
      HW_1913P1_EO_Multiturn_1 { ExternalAccessible := 'False'; ExternalVisible := 'False'; ExternalWritable := 'False'} : HW_SUBMODULE := 938;   // "1913P1~EO_Multiturn_1"
      HW_1913P1_Telegram_81_DI_DO { ExternalAccessible := 'False'; ExternalVisible := 'False'; ExternalWritable := 'False'} : HW_SUBMODULE := 939;   // "1913P1_Telegram_81~DI_DO"
      HW_1913P1_EO_Multiturn_1_Parameter_Access_Point { ExternalAccessible := 'False'; ExternalVisible := 'False'; ExternalWritable := 'False'} : HW_SUBMODULE := 940;   // "1913P1~EO_Multiturn_1~Parameter_Access_Point"
      HW_1908P1_Proxy { ExternalAccessible := 'False'; ExternalVisible := 'False'; ExternalWritable := 'False'} : HW_SUBMODULE := 943;   // "1908P1~Proxy"
      HW_1908P1_IODevice { ExternalAccessible := 'False'; ExternalVisible := 'False'; ExternalWritable := 'False'} : HW_DEVICE := 941;   // "1908P1~IODevice"
      HW_1908P1_Interface { ExternalAccessible := 'False'; ExternalVisible := 'False'; ExternalWritable := 'False'} : HW_INTERFACE := 944;   // "1908P1~Interface"
      HW_1908P1_Interface_Port_1 { ExternalAccessible := 'False'; ExternalVisible := 'False'; ExternalWritable := 'False'} : HW_INTERFACE := 945;   // "1908P1~Interface~Port_1"
      HW_1908P1_Interface_Port_2 { ExternalAccessible := 'False'; ExternalVisible := 'False'; ExternalWritable := 'False'} : HW_INTERFACE := 946;   // "1908P1~Interface~Port_2"
      HW_1908P1_Head { ExternalAccessible := 'False'; ExternalVisible := 'False'; ExternalWritable := 'False'} : HW_SUBMODULE := 947;   // "1908P1~Head"
      HW_1908P1_EO_Multiturn_1 { ExternalAccessible := 'False'; ExternalVisible := 'False'; ExternalWritable := 'False'} : HW_SUBMODULE := 948;   // "1908P1~EO_Multiturn_1"
      HW_1908P1_Telegram_81_DI_DO { ExternalAccessible := 'False'; ExternalVisible := 'False'; ExternalWritable := 'False'} : HW_SUBMODULE := 949;   // "1908P1_Telegram_81~DI_DO"
      HW_1908P1_EO_Multiturn_1_Parameter_Access_Point { ExternalAccessible := 'False'; ExternalVisible := 'False'; ExternalWritable := 'False'} : HW_SUBMODULE := 950;   // "1908P1~EO_Multiturn_1~Parameter_Access_Point"
      HW_1088P1_Proxy { ExternalAccessible := 'False'; ExternalVisible := 'False'; ExternalWritable := 'False'} : HW_SUBMODULE := 776;   // "1088P1~Proxy"
      HW_1088P1_IODevice { ExternalAccessible := 'False'; ExternalVisible := 'False'; ExternalWritable := 'False'} : HW_DEVICE := 774;   // "1088P1~IODevice"
      HW_1088P1_Interface { ExternalAccessible := 'False'; ExternalVisible := 'False'; ExternalWritable := 'False'} : HW_INTERFACE := 777;   // "1088P1~Interface"
      HW_1088P1_Interface_Port_1 { ExternalAccessible := 'False'; ExternalVisible := 'False'; ExternalWritable := 'False'} : HW_INTERFACE := 778;   // "1088P1~Interface~Port_1"
      HW_1088P1_Interface_Port_2 { ExternalAccessible := 'False'; ExternalVisible := 'False'; ExternalWritable := 'False'} : HW_INTERFACE := 779;   // "1088P1~Interface~Port_2"
      HW_1088P1_Head { ExternalAccessible := 'False'; ExternalVisible := 'False'; ExternalWritable := 'False'} : HW_SUBMODULE := 780;   // "1088P1~Head"
      HW_1088P1_EO_Multiturn_1 { ExternalAccessible := 'False'; ExternalVisible := 'False'; ExternalWritable := 'False'} : HW_SUBMODULE := 781;   // "1088P1~EO_Multiturn_1"
      HW_1088P1_Telegram_81_DI_DO { ExternalAccessible := 'False'; ExternalVisible := 'False'; ExternalWritable := 'False'} : HW_SUBMODULE := 782;   // "1088P1_Telegram_81~DI_DO"
      HW_1088P1_EO_Multiturn_1_Parameter_Access_Point { ExternalAccessible := 'False'; ExternalVisible := 'False'; ExternalWritable := 'False'} : HW_SUBMODULE := 783;   // "1088P1~EO_Multiturn_1~Parameter_Access_Point"
      HW_1074P1_Proxy { ExternalAccessible := 'False'; ExternalVisible := 'False'; ExternalWritable := 'False'} : HW_SUBMODULE := 796;   // "1074P1~Proxy"
      HW_1074P1_IODevice { ExternalAccessible := 'False'; ExternalVisible := 'False'; ExternalWritable := 'False'} : HW_DEVICE := 794;   // "1074P1~IODevice"
      HW_1074P1_Interface { ExternalAccessible := 'False'; ExternalVisible := 'False'; ExternalWritable := 'False'} : HW_INTERFACE := 797;   // "1074P1~Interface"
      HW_1074P1_Interface_Port_1 { ExternalAccessible := 'False'; ExternalVisible := 'False'; ExternalWritable := 'False'} : HW_INTERFACE := 798;   // "1074P1~Interface~Port_1"
      HW_1074P1_Interface_Port_2 { ExternalAccessible := 'False'; ExternalVisible := 'False'; ExternalWritable := 'False'} : HW_INTERFACE := 799;   // "1074P1~Interface~Port_2"
      HW_1074P1_Head { ExternalAccessible := 'False'; ExternalVisible := 'False'; ExternalWritable := 'False'} : HW_SUBMODULE := 800;   // "1074P1~Head"
      HW_1074P1_EO_Multiturn_1 { ExternalAccessible := 'False'; ExternalVisible := 'False'; ExternalWritable := 'False'} : HW_SUBMODULE := 801;   // "1074P1~EO_Multiturn_1"
      HW_1074P1_Telegram_81_DI_DO { ExternalAccessible := 'False'; ExternalVisible := 'False'; ExternalWritable := 'False'} : HW_SUBMODULE := 802;   // "1074P1_Telegram_81~DI_DO"
      HW_1074P1_EO_Multiturn_1_Parameter_Access_Point { ExternalAccessible := 'False'; ExternalVisible := 'False'; ExternalWritable := 'False'} : HW_SUBMODULE := 803;   // "1074P1~EO_Multiturn_1~Parameter_Access_Point"
      HW_1903P1_Proxy { ExternalAccessible := 'False'; ExternalVisible := 'False'; ExternalWritable := 'False'} : HW_SUBMODULE := 953;   // "1903P1~Proxy"
      HW_1903P1_IODevice { ExternalAccessible := 'False'; ExternalVisible := 'False'; ExternalWritable := 'False'} : HW_DEVICE := 951;   // "1903P1~IODevice"
      HW_1903P1_Interface { ExternalAccessible := 'False'; ExternalVisible := 'False'; ExternalWritable := 'False'} : HW_INTERFACE := 954;   // "1903P1~Interface"
      HW_1903P1_Interface_Port_1 { ExternalAccessible := 'False'; ExternalVisible := 'False'; ExternalWritable := 'False'} : HW_INTERFACE := 955;   // "1903P1~Interface~Port_1"
      HW_1903P1_Interface_Port_2 { ExternalAccessible := 'False'; ExternalVisible := 'False'; ExternalWritable := 'False'} : HW_INTERFACE := 956;   // "1903P1~Interface~Port_2"
      HW_1903P1_Head { ExternalAccessible := 'False'; ExternalVisible := 'False'; ExternalWritable := 'False'} : HW_SUBMODULE := 957;   // "1903P1~Head"
      HW_1903P1_EO_Multiturn_1 { ExternalAccessible := 'False'; ExternalVisible := 'False'; ExternalWritable := 'False'} : HW_SUBMODULE := 958;   // "1903P1~EO_Multiturn_1"
      HW_1903P1_Telegram_81_DI_DO { ExternalAccessible := 'False'; ExternalVisible := 'False'; ExternalWritable := 'False'} : HW_SUBMODULE := 959;   // "1903P1_Telegram_81~DI_DO"
      HW_1903P1_EO_Multiturn_1_Parameter_Access_Point { ExternalAccessible := 'False'; ExternalVisible := 'False'; ExternalWritable := 'False'} : HW_SUBMODULE := 960;   // "1903P1~EO_Multiturn_1~Parameter_Access_Point"
      HW_1143P1_Proxy { ExternalAccessible := 'False'; ExternalVisible := 'False'; ExternalWritable := 'False'} : HW_SUBMODULE := 806;   // "1143P1~Proxy"
      HW_1143P1_IODevice { ExternalAccessible := 'False'; ExternalVisible := 'False'; ExternalWritable := 'False'} : HW_DEVICE := 804;   // "1143P1~IODevice"
      HW_1143P1_Interface { ExternalAccessible := 'False'; ExternalVisible := 'False'; ExternalWritable := 'False'} : HW_INTERFACE := 807;   // "1143P1~Interface"
      HW_1143P1_Interface_Port_1 { ExternalAccessible := 'False'; ExternalVisible := 'False'; ExternalWritable := 'False'} : HW_INTERFACE := 808;   // "1143P1~Interface~Port_1"
      HW_1143P1_Interface_Port_2 { ExternalAccessible := 'False'; ExternalVisible := 'False'; ExternalWritable := 'False'} : HW_INTERFACE := 809;   // "1143P1~Interface~Port_2"
      HW_1143P1_Head { ExternalAccessible := 'False'; ExternalVisible := 'False'; ExternalWritable := 'False'} : HW_SUBMODULE := 810;   // "1143P1~Head"
      HW_1143P1_EO_Multiturn_1 { ExternalAccessible := 'False'; ExternalVisible := 'False'; ExternalWritable := 'False'} : HW_SUBMODULE := 811;   // "1143P1~EO_Multiturn_1"
      HW_1143P1_Telegram_81_DI_DO { ExternalAccessible := 'False'; ExternalVisible := 'False'; ExternalWritable := 'False'} : HW_SUBMODULE := 812;   // "1143P1_Telegram_81~DI_DO"
      HW_1143P1_EO_Multiturn_1_Parameter_Access_Point { ExternalAccessible := 'False'; ExternalVisible := 'False'; ExternalWritable := 'False'} : HW_SUBMODULE := 813;   // "1143P1~EO_Multiturn_1~Parameter_Access_Point"
      HW_1138P1_Proxy { ExternalAccessible := 'False'; ExternalVisible := 'False'; ExternalWritable := 'False'} : HW_SUBMODULE := 816;   // "1138P1~Proxy"
      HW_1138P1_IODevice { ExternalAccessible := 'False'; ExternalVisible := 'False'; ExternalWritable := 'False'} : HW_DEVICE := 814;   // "1138P1~IODevice"
      HW_1138P1_Interface { ExternalAccessible := 'False'; ExternalVisible := 'False'; ExternalWritable := 'False'} : HW_INTERFACE := 817;   // "1138P1~Interface"
      HW_1138P1_Interface_Port_1 { ExternalAccessible := 'False'; ExternalVisible := 'False'; ExternalWritable := 'False'} : HW_INTERFACE := 818;   // "1138P1~Interface~Port_1"
      HW_1138P1_Interface_Port_2 { ExternalAccessible := 'False'; ExternalVisible := 'False'; ExternalWritable := 'False'} : HW_INTERFACE := 819;   // "1138P1~Interface~Port_2"
      HW_1138P1_Head { ExternalAccessible := 'False'; ExternalVisible := 'False'; ExternalWritable := 'False'} : HW_SUBMODULE := 820;   // "1138P1~Head"
      HW_1138P1_EO_Multiturn_1 { ExternalAccessible := 'False'; ExternalVisible := 'False'; ExternalWritable := 'False'} : HW_SUBMODULE := 821;   // "1138P1~EO_Multiturn_1"
      HW_1138P1_Telegram_81_DI_DO { ExternalAccessible := 'False'; ExternalVisible := 'False'; ExternalWritable := 'False'} : HW_SUBMODULE := 822;   // "1138P1_Telegram_81~DI_DO"
      HW_1138P1_EO_Multiturn_1_Parameter_Access_Point { ExternalAccessible := 'False'; ExternalVisible := 'False'; ExternalWritable := 'False'} : HW_SUBMODULE := 823;   // "1138P1~EO_Multiturn_1~Parameter_Access_Point"
      HW_2264P1_Proxy { ExternalAccessible := 'False'; ExternalVisible := 'False'; ExternalWritable := 'False'} : HW_SUBMODULE := 963;   // "2264P1~Proxy"
      HW_2264P1_IODevice { ExternalAccessible := 'False'; ExternalVisible := 'False'; ExternalWritable := 'False'} : HW_DEVICE := 961;   // "2264P1~IODevice"
      HW_2264P1_Interface { ExternalAccessible := 'False'; ExternalVisible := 'False'; ExternalWritable := 'False'} : HW_INTERFACE := 964;   // "2264P1~Interface"
      HW_2264P1_Interface_Port_1 { ExternalAccessible := 'False'; ExternalVisible := 'False'; ExternalWritable := 'False'} : HW_INTERFACE := 965;   // "2264P1~Interface~Port_1"
      HW_2264P1_Interface_Port_2 { ExternalAccessible := 'False'; ExternalVisible := 'False'; ExternalWritable := 'False'} : HW_INTERFACE := 966;   // "2264P1~Interface~Port_2"
      HW_2264P1_Head { ExternalAccessible := 'False'; ExternalVisible := 'False'; ExternalWritable := 'False'} : HW_SUBMODULE := 967;   // "2264P1~Head"
      HW_2264P1_EO_Multiturn_1 { ExternalAccessible := 'False'; ExternalVisible := 'False'; ExternalWritable := 'False'} : HW_SUBMODULE := 968;   // "2264P1~EO_Multiturn_1"
      HW_2264P1_Telegram_81_DI_DO { ExternalAccessible := 'False'; ExternalVisible := 'False'; ExternalWritable := 'False'} : HW_SUBMODULE := 969;   // "2264P1_Telegram_81~DI_DO"
      HW_2264P1_EO_Multiturn_1_Parameter_Access_Point { ExternalAccessible := 'False'; ExternalVisible := 'False'; ExternalWritable := 'False'} : HW_SUBMODULE := 970;   // "2264P1~EO_Multiturn_1~Parameter_Access_Point"
      HW_1124P1_Proxy { ExternalAccessible := 'False'; ExternalVisible := 'False'; ExternalWritable := 'False'} : HW_SUBMODULE := 836;   // "1124P1~Proxy"
      HW_1124P1_IODevice { ExternalAccessible := 'False'; ExternalVisible := 'False'; ExternalWritable := 'False'} : HW_DEVICE := 834;   // "1124P1~IODevice"
      HW_1124P1_Interface { ExternalAccessible := 'False'; ExternalVisible := 'False'; ExternalWritable := 'False'} : HW_INTERFACE := 837;   // "1124P1~Interface"
      HW_1124P1_Interface_Port_1 { ExternalAccessible := 'False'; ExternalVisible := 'False'; ExternalWritable := 'False'} : HW_INTERFACE := 838;   // "1124P1~Interface~Port_1"
      HW_1124P1_Interface_Port_2 { ExternalAccessible := 'False'; ExternalVisible := 'False'; ExternalWritable := 'False'} : HW_INTERFACE := 839;   // "1124P1~Interface~Port_2"
      HW_1124P1_Head { ExternalAccessible := 'False'; ExternalVisible := 'False'; ExternalWritable := 'False'} : HW_SUBMODULE := 840;   // "1124P1~Head"
      HW_1124P1_EO_Multiturn_1 { ExternalAccessible := 'False'; ExternalVisible := 'False'; ExternalWritable := 'False'} : HW_SUBMODULE := 841;   // "1124P1~EO_Multiturn_1"
      HW_1124P1_Telegram_81_DI_DO { ExternalAccessible := 'False'; ExternalVisible := 'False'; ExternalWritable := 'False'} : HW_SUBMODULE := 842;   // "1124P1_Telegram_81~DI_DO"
      HW_1124P1_EO_Multiturn_1_Parameter_Access_Point { ExternalAccessible := 'False'; ExternalVisible := 'False'; ExternalWritable := 'False'} : HW_SUBMODULE := 843;   // "1124P1~EO_Multiturn_1~Parameter_Access_Point"
      HW_2284P1_Proxy { ExternalAccessible := 'False'; ExternalVisible := 'False'; ExternalWritable := 'False'} : HW_SUBMODULE := 973;   // "2284P1~Proxy"
      HW_2284P1_IODevice { ExternalAccessible := 'False'; ExternalVisible := 'False'; ExternalWritable := 'False'} : HW_DEVICE := 971;   // "2284P1~IODevice"
      HW_2284P1_Interface { ExternalAccessible := 'False'; ExternalVisible := 'False'; ExternalWritable := 'False'} : HW_INTERFACE := 974;   // "2284P1~Interface"
      HW_2284P1_Interface_Port_1 { ExternalAccessible := 'False'; ExternalVisible := 'False'; ExternalWritable := 'False'} : HW_INTERFACE := 975;   // "2284P1~Interface~Port_1"
      HW_2284P1_Interface_Port_2 { ExternalAccessible := 'False'; ExternalVisible := 'False'; ExternalWritable := 'False'} : HW_INTERFACE := 976;   // "2284P1~Interface~Port_2"
      HW_2284P1_Head { ExternalAccessible := 'False'; ExternalVisible := 'False'; ExternalWritable := 'False'} : HW_SUBMODULE := 977;   // "2284P1~Head"
      HW_2284P1_EO_Multiturn_1 { ExternalAccessible := 'False'; ExternalVisible := 'False'; ExternalWritable := 'False'} : HW_SUBMODULE := 978;   // "2284P1~EO_Multiturn_1"
      HW_2284P1_Telegram_81_DI_DO { ExternalAccessible := 'False'; ExternalVisible := 'False'; ExternalWritable := 'False'} : HW_SUBMODULE := 979;   // "2284P1_Telegram_81~DI_DO"
      HW_2284P1_EO_Multiturn_1_Parameter_Access_Point { ExternalAccessible := 'False'; ExternalVisible := 'False'; ExternalWritable := 'False'} : HW_SUBMODULE := 980;   // "2284P1~EO_Multiturn_1~Parameter_Access_Point"
      HW_694P1_Proxy { ExternalAccessible := 'False'; ExternalVisible := 'False'; ExternalWritable := 'False'} : HW_SUBMODULE := 846;   // "694P1~Proxy"
      HW_694P1_IODevice { ExternalAccessible := 'False'; ExternalVisible := 'False'; ExternalWritable := 'False'} : HW_DEVICE := 844;   // "694P1~IODevice"
      HW_694P1_Interface { ExternalAccessible := 'False'; ExternalVisible := 'False'; ExternalWritable := 'False'} : HW_INTERFACE := 847;   // "694P1~Interface"
      HW_694P1_Interface_Port_1 { ExternalAccessible := 'False'; ExternalVisible := 'False'; ExternalWritable := 'False'} : HW_INTERFACE := 848;   // "694P1~Interface~Port_1"
      HW_694P1_Interface_Port_2 { ExternalAccessible := 'False'; ExternalVisible := 'False'; ExternalWritable := 'False'} : HW_INTERFACE := 849;   // "694P1~Interface~Port_2"
      HW_694P1_Head { ExternalAccessible := 'False'; ExternalVisible := 'False'; ExternalWritable := 'False'} : HW_SUBMODULE := 850;   // "694P1~Head"
      HW_694P1_EO_Multiturn_1 { ExternalAccessible := 'False'; ExternalVisible := 'False'; ExternalWritable := 'False'} : HW_SUBMODULE := 851;   // "694P1~EO_Multiturn_1"
      HW_694P1_Telegram_81_DI_DO { ExternalAccessible := 'False'; ExternalVisible := 'False'; ExternalWritable := 'False'} : HW_SUBMODULE := 852;   // "694P1_Telegram_81~DI_DO"
      HW_694P1_EO_Multiturn_1_Parameter_Access_Point { ExternalAccessible := 'False'; ExternalVisible := 'False'; ExternalWritable := 'False'} : HW_SUBMODULE := 853;   // "694P1~EO_Multiturn_1~Parameter_Access_Point"
      HW_2354P1_Proxy { ExternalAccessible := 'False'; ExternalVisible := 'False'; ExternalWritable := 'False'} : HW_SUBMODULE := 983;   // "2354P1~Proxy"
      HW_2354P1_IODevice { ExternalAccessible := 'False'; ExternalVisible := 'False'; ExternalWritable := 'False'} : HW_DEVICE := 981;   // "2354P1~IODevice"
      HW_2354P1_Interface { ExternalAccessible := 'False'; ExternalVisible := 'False'; ExternalWritable := 'False'} : HW_INTERFACE := 984;   // "2354P1~Interface"
      HW_2354P1_Interface_Port_1 { ExternalAccessible := 'False'; ExternalVisible := 'False'; ExternalWritable := 'False'} : HW_INTERFACE := 985;   // "2354P1~Interface~Port_1"
      HW_2354P1_Interface_Port_2 { ExternalAccessible := 'False'; ExternalVisible := 'False'; ExternalWritable := 'False'} : HW_INTERFACE := 986;   // "2354P1~Interface~Port_2"
      HW_2354P1_Head { ExternalAccessible := 'False'; ExternalVisible := 'False'; ExternalWritable := 'False'} : HW_SUBMODULE := 987;   // "2354P1~Head"
      HW_2354P1_EO_Multiturn_1 { ExternalAccessible := 'False'; ExternalVisible := 'False'; ExternalWritable := 'False'} : HW_SUBMODULE := 988;   // "2354P1~EO_Multiturn_1"
      HW_2354P1_Telegram_81_DI_DO { ExternalAccessible := 'False'; ExternalVisible := 'False'; ExternalWritable := 'False'} : HW_SUBMODULE := 989;   // "2354P1_Telegram_81~DI_DO"
      HW_2354P1_EO_Multiturn_1_Parameter_Access_Point { ExternalAccessible := 'False'; ExternalVisible := 'False'; ExternalWritable := 'False'} : HW_SUBMODULE := 990;   // "2354P1~EO_Multiturn_1~Parameter_Access_Point"
      HW_894P1_Proxy { ExternalAccessible := 'False'; ExternalVisible := 'False'; ExternalWritable := 'False'} : HW_SUBMODULE := 856;   // "894P1~Proxy"
      HW_894P1_IODevice { ExternalAccessible := 'False'; ExternalVisible := 'False'; ExternalWritable := 'False'} : HW_DEVICE := 854;   // "894P1~IODevice"
      HW_894P1_Interface { ExternalAccessible := 'False'; ExternalVisible := 'False'; ExternalWritable := 'False'} : HW_INTERFACE := 857;   // "894P1~Interface"
      HW_894P1_Interface_Port_1 { ExternalAccessible := 'False'; ExternalVisible := 'False'; ExternalWritable := 'False'} : HW_INTERFACE := 858;   // "894P1~Interface~Port_1"
      HW_894P1_Interface_Port_2 { ExternalAccessible := 'False'; ExternalVisible := 'False'; ExternalWritable := 'False'} : HW_INTERFACE := 859;   // "894P1~Interface~Port_2"
      HW_894P1_Head { ExternalAccessible := 'False'; ExternalVisible := 'False'; ExternalWritable := 'False'} : HW_SUBMODULE := 860;   // "894P1~Head"
      HW_894P1_EO_Multiturn_1 { ExternalAccessible := 'False'; ExternalVisible := 'False'; ExternalWritable := 'False'} : HW_SUBMODULE := 861;   // "894P1~EO_Multiturn_1"
      HW_894P1_Telegram_81_DI_DO { ExternalAccessible := 'False'; ExternalVisible := 'False'; ExternalWritable := 'False'} : HW_SUBMODULE := 862;   // "894P1_Telegram_81~DI_DO"
      HW_894P1_EO_Multiturn_1_Parameter_Access_Point { ExternalAccessible := 'False'; ExternalVisible := 'False'; ExternalWritable := 'False'} : HW_SUBMODULE := 863;   // "894P1~EO_Multiturn_1~Parameter_Access_Point"
      HW_2374P1_Proxy { ExternalAccessible := 'False'; ExternalVisible := 'False'; ExternalWritable := 'False'} : HW_SUBMODULE := 993;   // "2374P1~Proxy"
      HW_2374P1_IODevice { ExternalAccessible := 'False'; ExternalVisible := 'False'; ExternalWritable := 'False'} : HW_DEVICE := 991;   // "2374P1~IODevice"
      HW_2374P1_Interface { ExternalAccessible := 'False'; ExternalVisible := 'False'; ExternalWritable := 'False'} : HW_INTERFACE := 994;   // "2374P1~Interface"
